// TwinCAT 3 PLC project ExternControl
// ProgramVersion: 3.1.4026.26
// libraries:
//   Tc2_Standard, * (Beckhoff Automation GmbH)
//   Tc2_System, * (Beckhoff Automation GmbH)
//   Tc2_Utilities, * (Beckhoff Automation GmbH)
// project tree:
//   APPLICATION/DISPENSER/types/ ST_DISPENSER_AXIS_PARAMETER.TcDUT, ST_DISPENSER_JOB_PARAMETER.TcDUT, ST_DISPENSER_PARAMETER.TcDUT, ST_DISPENSER_VALVES.TcDUT
//   APPLICATION/ GVL_APPLICATION.TcGVL
//   APPLICATION/JOB_CONTROL/ fb_JobBase.TcPOU, fb_JobCtrl.TcPOU
//   APPLICATION/JOB_CONTROL/types/ E_JOB_CTRL.TcDUT, E_JOB_STATE.TcDUT, E_M_FUNC.TcDUT, E_R_PARAMETER.TcDUT, E_JOB_CHECK.TcDUT, ST_AXIS_GROUP_INFO.TcDUT, ST_JOB_CTRL.TcDUT, ST_JOB_PARAMETER.TcDUT, ST_JOB_STATE.TcDUT, ST_PROG_PARAMETER.TcDUT, ST_R_ProgParameter.TcDUT, ST_TUPEL_XYZ.TcDUT
//   / GlobalTextList.TcGTLO, MAIN.TcPOU, PlcTask.TcTTO (not stored), Visualization Manager.TcVMO (not stored)
//   MAPPING/ MAPPING_out.TcPOU, MAPPING_in.TcPOU
//   MAPPING/types/ U_AXIS_CTRL.TcDUT (not stored), U_AXIS_GEAR_IN.TcDUT (not stored), U_AXIS_HOMING.TcDUT, U_AXIS_INFO.TcDUT, U_AXIS_MOTION_OPTIONS.TcDUT (not stored), U_AXIS_MOVE_DATA.TcDUT, U_AXIS_NC_PARAMETER_RD.TcDUT (not stored), U_AXIS_NC_PARAMETER_WRT.TcDUT (not stored), U_AXIS_STATE.TcDUT, U_CAM_CTRL.TcDUT, U_CAM_DATA.TcDUT, U_CAM_INFO.TcDUT (not stored), U_CAM_STATE.TcDUT, U_NCI_AXIS_ID_GROUP.TcDUT, U_NCI_CTRL.TcDUT, U_NCI_INDEX_GROUP.TcDUT (not stored), U_NCI_R_PARAMETER_I.TcDUT, U_NCI_R_PARAMETER_Q.TcDUT, U_NCI_STATE.TcDUT (not stored), U_TOUCH_PROBE_CTRL.TcDUT (not stored), U_TOUCH_PROBE_STATE.TcDUT, U_TRIGGER_CTRL.TcDUT (not stored), U_TRIGGER_STATE.TcDUT
//   PLC_MOTION/CAM/ GVL_CAM.TcGVL
//   PLC_MOTION/CAM/types/ ST_CAM_CTRL.TcDUT (not stored), ST_CAM_DATA.TcDUT, ST_CAM_INFO.TcDUT, ST_CAM_OPTIONS.TcDUT, ST_CAM_READ_VALUES_PARAMETER.TcDUT (not stored), ST_CAM_SCALING_DATA.TcDUT (not stored), ST_CAM_STATE.TcDUT, ST_MOTION_FUNCTION.TcDUT (not stored), ST_MOTION_FUNCTION_POINT.TcDUT
//   PLC_MOTION/FUNCTIONS/ GVL_FUNCTIONS.TcGVL
//   PLC_MOTION/FUNCTIONS/TOUCH_PROBE/types/ ST_2BIT.TcDUT, ST_CTRL_TOUCH_PROBE.TcDUT (not stored), ST_DC_Input.TcDUT (not stored), ST_MTI_INPUT.TcDUT (not stored), ST_MTI_STATUS.TcDUT (not stored), ST_STATE_TOUCH_PROBE.TcDUT (not stored)
//   PLC_MOTION/FUNCTIONS/TRIGGER_BOX/types/ ST_CTRL_TRIGGER.TcDUT (not stored), ST_DC_Output.TcDUT, ST_DC_State.TcDUT, ST_STATE_TRIGGER.TcDUT, T_TriggerControlBits.TcDUT
//   PLC_MOTION/NCI/ GVL_NCI.TcGVL
//   PLC_MOTION/NCI/types/ E_NCI_CHANNEL_ERROR.TcDUT, E_NCI_CTRL.TcDUT, E_NCI_INTERPRETER_STATE.TcDUT (not stored), E_NCI_STATE.TcDUT, ST_3D_Group.TcDUT (not stored), ST_Index_Group.TcDUT, ST_Interface_Group.TcDUT, ST_NciChannel_Ref.TcDUT (not stored), ST_NCI_CTRL.TcDUT (not stored), ST_NCI_M_FUNC.TcDUT (not stored), ST_NCI_STATE.TcDUT, ST_R_Parameter.TcDUT (not stored)
//   PLC_MOTION/NC_PTP/ GVL_AXIS.TcGVL (not stored)
//   PLC_MOTION/NC_PTP/types/axis/ E_AxisEncoderType.TcDUT (not stored), ST_HomeParams.TcDUT (not stored), ST_HomingOptionsExt.TcDUT (not stored)
//   PLC_MOTION/NC_PTP/types/control/ E_AXIS_CTRL.TcDUT, E_AXIS_STATE.TcDUT, ST_AXIS_CTRL.TcDUT (not stored), ST_AXIS_INFO.TcDUT (not stored), ST_AXIS_STATE.TcDUT, ST_GEAR_IN.TcDUT (not stored), ST_HOMING.TcDUT, ST_MOTION_OPTIONS.TcDUT, ST_MOVE_DATA.TcDUT (not stored), ST_NC_PARAMETER.TcDUT
//   PLC_MOTION/_GVL/ PLC_CONSTANT.TcGVL (not stored)
//   XTS_TRANSPORT/ GVL_XTS_CONSTANTS.TcGVL
//   _DUT/ f_GetProgress.TcPOU (not stored), f_GetState.TcPOU (not stored), E_CHECK_STATE.TcDUT (not stored), E_PROGRESS.TcDUT (not stored)
//   _MSG/class/ fb_LocalTime.TcPOU, fb_MessageData.TcPOU, fb_MessageDataCtrl.TcPOU
//   _MSG/ f_MessageSet.TcPOU, GVL_MSG_AXIS.TcGVL, GVL_MSG_XTS.TcGVL, I_MessageData.TcIO
//   _MSG/types/ e_Device.TcDUT, E_MessageType.TcDUT, E_MESSAGE_BATCH.TcDUT (not stored), E_MESSAGE_CHECK.TcDUT, E_MESSAGE_CTRL.TcDUT (not stored), E_MESSAGE_FLOW.TcDUT, E_MESSAGE_STATE.TcDUT (not stored), e_Subdevice.TcDUT, ST_Message.TcDUT (not stored), ST_MESSAGE_CTRL.TcDUT (not stored), ST_MESSAGE_STATE.TcDUT (not stored), TL_E_MESSAGETYPE.TcTLO
//   _XML/Configuration/ fb_Configuration.TcPOU
//   _XML/Configuration/types/ ST_Configuration.TcDUT, ST_CONFIG_DISPENSER.TcDUT, ST_CONFIG_JOBS.TcDUT, ST_CONFIG_PORTAL.TcDUT
//   _XML/ fb_XmlBase.TcPOU
//   _XML/types/ E_DATA_CHECK.TcDUT (not stored), E_DATA_CTRL.TcDUT (not stored), E_DATA_STATE.TcDUT (not stored), fb_XmlRead.TcPOU (not stored), fb_XmlWrite.TcPOU (not stored), ST_DATA_CTRL.TcDUT (not stored), ST_DATA_STATE.TcDUT (not stored)
// real-time tasks:
//   TASK PlcTask: cycle T#1ms, priority 20, ADS port 350
// motion (NC):
//   TASK NC-Task 1 SAF: cycle T#2ms, priority 4, ADS port 501
//   TASK NC-Task 1 SVB: cycle T#10ms, priority 8, ADS port 511
//   AXIS AxisX (id 1)
//     OtherSettings: AllowMotionCmdToSlave=true
//     encoder EncType=1
//     drive DrvType=5
//       Analog: TorqueSetpointScale=10, ScaleFactorActTorque=0.1
//       TimeComp: TaskDelayCycles=1
//     controller CtrType=1
//       CtrPara: PriorControlFactor=1
//         Observer: BandWidth=20
//   AXIS AxisY (id 2)
//     OtherSettings: AllowMotionCmdToSlave=true
//     encoder EncType=1
//     drive DrvType=5
//       Analog: TorqueSetpointScale=10, ScaleFactorActTorque=0.1
//       TimeComp: TaskDelayCycles=1
//     controller CtrType=1
//       CtrPara: PriorControlFactor=1
//         Observer: BandWidth=20
//   AXIS AxisZ (id 3)
//     OtherSettings: AllowMotionCmdToSlave=true
//     encoder EncType=1
//     drive DrvType=5
//       Analog: TorqueSetpointScale=10, ScaleFactorActTorque=0.1
//       TimeComp: TaskDelayCycles=1
//     controller CtrType=1
//       CtrPara: PriorControlFactor=1
//         Observer: BandWidth=20
//   AXIS Dos_A1 (id 4)
//     OtherSettings: AllowMotionCmdToSlave=true
//     encoder EncType=1
//     drive DrvType=5
//       Analog: TorqueSetpointScale=10, ScaleFactorActTorque=0.1
//       TimeComp: TaskDelayCycles=1
//     controller CtrType=1
//       CtrPara: PriorControlFactor=1
//         Observer: BandWidth=20
//   AXIS Dos_A2 (id 5)
//     OtherSettings: AllowMotionCmdToSlave=true
//     encoder EncType=1
//     drive DrvType=5
//       Analog: TorqueSetpointScale=10, ScaleFactorActTorque=0.1
//       TimeComp: TaskDelayCycles=1
//     controller CtrType=1
//       CtrPara: PriorControlFactor=1
//         Observer: BandWidth=20
//   AXIS Axis 6 (id 6)
//     OtherSettings: AllowMotionCmdToSlave=true
//     encoder EncType=1
//     drive DrvType=5
//       Analog: TorqueSetpointScale=10, ScaleFactorActTorque=0.1
//       TimeComp: TaskDelayCycles=1
//     controller CtrType=1
//       CtrPara: PriorControlFactor=1
//         Observer: BandWidth=20
// variable links:
//   ExternControl/ExternControl Instance <-> PLC_MOTION/PLC_MOTION Instance
//     PlcTask Inputs/MAIN.eInitPlcMotion <-> PlcTask Outputs/MAIN_AXIS.eInit
//     PlcTask Inputs/MAPPING_in.AxisInfo.byState <-> PlcTask Outputs/MAPPING_AXIS_out.AxisInfo.byState
//     PlcTask Inputs/MAPPING_in.AxisParameterRd.byState <-> PlcTask Outputs/MAPPING_AXIS_out.AxisParameterOut.byState
//     PlcTask Inputs/MAPPING_in.AxisState.byState <-> PlcTask Outputs/MAPPING_AXIS_out.AxisState.byState
//     PlcTask Inputs/MAPPING_in.CamInfo.byState <-> PlcTask Outputs/MAPPING_AXIS_out.CamInfo.byState
//     PlcTask Inputs/MAPPING_in.CamState.byState <-> PlcTask Outputs/MAPPING_AXIS_out.CamState.byState
//     PlcTask Inputs/MAPPING_in.NciRparameters.byState <-> PlcTask Outputs/MAPPING_AXIS_out.NciRparameters.byCtrl
//     PlcTask Inputs/MAPPING_in.NciState.byState <-> PlcTask Outputs/MAPPING_AXIS_out.NciState.byState
//     PlcTask Inputs/MAPPING_in.TouchState.byState <-> PlcTask Outputs/MAPPING_AXIS_out.TouchProbeState.byState
//     PlcTask Inputs/MAPPING_in.TriggerState.byState <-> PlcTask Outputs/MAPPING_AXIS_out.TriggerState.byState
//     PlcTask Outputs/MAPPING_out.AxisCtrl.byCtrl <-> PlcTask Inputs/MAPPING_AXIS_in.AxisCtrl.byCtrl
//     PlcTask Outputs/MAPPING_out.AxisGearInData.byCtrl <-> PlcTask Inputs/MAPPING_AXIS_in.AxisGearInData.byCtrl
//     PlcTask Outputs/MAPPING_out.AxisHoming.byCtrl <-> PlcTask Inputs/MAPPING_AXIS_in.AxisHoming.byCtrl
//     PlcTask Outputs/MAPPING_out.AxisMotionOptions.byCtrl <-> PlcTask Inputs/MAPPING_AXIS_in.AxisMotionOptions.byCtrl
//     PlcTask Outputs/MAPPING_out.AxisMoveData.byCtrl <-> PlcTask Inputs/MAPPING_AXIS_in.AxisMoveData.byCtrl
//     PlcTask Outputs/MAPPING_out.AxisParameterWrt.byCtrl <-> PlcTask Inputs/MAPPING_AXIS_in.AxisParameterIn.byCtrl
//     PlcTask Outputs/MAPPING_out.CamCtrl.byCtrl <-> PlcTask Inputs/MAPPING_AXIS_in.CamControl.byCtrl
//     PlcTask Outputs/MAPPING_out.CamData.byCtrl <-> PlcTask Inputs/MAPPING_AXIS_in.CamData.byCtrl
//     PlcTask Outputs/MAPPING_out.NciAxisGroup.byCtrl <-> PlcTask Inputs/MAPPING_AXIS_in.NciAxisGroup.byCtrl
//     PlcTask Outputs/MAPPING_out.NciControl.byCtrl <-> PlcTask Inputs/MAPPING_AXIS_in.NciControl.byCtrl[1]
//     PlcTask Outputs/MAPPING_out.NciRparameters.byCtrl <-> PlcTask Inputs/MAPPING_AXIS_in.NciRparameters.byCtrl
//     PlcTask Outputs/MAPPING_out.TouchCtrl.byCtrl <-> PlcTask Inputs/MAPPING_AXIS_in.TouchProbeControl.byCtrl
//     PlcTask Outputs/MAPPING_out.TriggerCtrl.byCtrl <-> PlcTask Inputs/MAPPING_AXIS_in.TriggerControl.byCtrl
//   PLC_MOTION/PLC_MOTION Instance <-> NC-Task 1 SAF/Axes/Axis 6
//     PlcTask Inputs/GVL_AXIS.AxisRef[6].NcToPlc <-> Outputs/ToPlc
//     PlcTask Outputs/GVL_AXIS.AxisRef[6].PlcToNc <-> Inputs/FromPlc
//   PLC_MOTION/PLC_MOTION Instance <-> NC-Task 1 SAF/Axes/AxisX
//     PlcTask Inputs/GVL_AXIS.AxisRef[1].NcToPlc <-> Outputs/ToPlc
//     PlcTask Outputs/GVL_AXIS.AxisRef[1].PlcToNc <-> Inputs/FromPlc
//   PLC_MOTION/PLC_MOTION Instance <-> NC-Task 1 SAF/Axes/AxisY
//     PlcTask Inputs/GVL_AXIS.AxisRef[2].NcToPlc <-> Outputs/ToPlc
//     PlcTask Outputs/GVL_AXIS.AxisRef[2].PlcToNc <-> Inputs/FromPlc
//   PLC_MOTION/PLC_MOTION Instance <-> NC-Task 1 SAF/Axes/AxisZ
//     PlcTask Inputs/GVL_AXIS.AxisRef[3].NcToPlc <-> Outputs/ToPlc
//     PlcTask Outputs/GVL_AXIS.AxisRef[3].PlcToNc <-> Inputs/FromPlc
//   PLC_MOTION/PLC_MOTION Instance <-> NC-Task 1 SAF/Axes/Dos_A1
//     PlcTask Inputs/GVL_AXIS.AxisRef[4].NcToPlc <-> Outputs/ToPlc
//     PlcTask Outputs/GVL_AXIS.AxisRef[4].PlcToNc <-> Inputs/FromPlc
//   PLC_MOTION/PLC_MOTION Instance <-> NC-Task 1 SAF/Axes/Dos_A2
//     PlcTask Inputs/GVL_AXIS.AxisRef[5].NcToPlc <-> Outputs/ToPlc
//     PlcTask Outputs/GVL_AXIS.AxisRef[5].PlcToNc <-> Inputs/FromPlc
//   PLC_MOTION/PLC_MOTION Instance <-> NC-Task 1 SAF/Channel XYZ
//     PlcTask Inputs/GVL_NCI.NciCtrl[1]._stChannelRef.NcToPlc <-> Outputs/ToPlc
//     PlcTask Outputs/GVL_NCI.NciCtrl[1]._stChannelRef.PlcToNc <-> Inputs/FromPlc

// ---- APPLICATION/DISPENSER/types/ST_DISPENSER_AXIS_PARAMETER.TcDUT
TYPE ST_DISPENSER_AXIS_PARAMETER :
STRUCT
  // configuration data for dispenser axis
  AxisIndex       : UINT;   // gfbAxisController[] index for PLC MOTION LAYER
  PistonDiameter  : LREAL :=   2.0;   // diameter for volume calc
  PistonArea      : LREAL :=  PI;     // (PistonDiameter/2)² * PI
  LimitUpper      : LREAL :=  10.0;   // upper limit of axis
  LimitLower      : LREAL :=   0.0;   // lower limit of axis
  LimitVelo       : LREAL :=  50.0;   // max dispensing velocity --> material constant
  LimitAccDec     : LREAL := 500.0;   // max dynamic --> material constant
END_STRUCT
END_TYPE

// ---- APPLICATION/DISPENSER/types/ST_DISPENSER_JOB_PARAMETER.TcDUT
TYPE ST_DISPENSER_JOB_PARAMETER :
STRUCT
  Volume    : LREAL := 10.0;      // [mm³]
  Velocity  : LREAL := 10.0;      // [mm³/s]
  AccDec    : LREAL := 100.0;     // [mm³/s²]
  tDelay    : TIME  := T#10MS;    // [ms]
END_STRUCT
END_TYPE

// ---- APPLICATION/DISPENSER/types/ST_DISPENSER_PARAMETER.TcDUT
TYPE ST_DISPENSER_PARAMETER :
STRUCT
  Component           : UINT  := 1;       // 1 or 2 component dispenser
  ValveInDelay        : TIME  := T#10MS;  // switch time for infeed valves  [ms]
  ValveOutDelay       : TIME  := T#10MS;  // switch time for outfeed valves [ms]

  AxisParameter       : ARRAY[1..GVL_APPLICATION.MAX_DISPENSER_COMPONENT] OF ST_DISPENSER_AXIS_PARAMETER;
END_STRUCT
END_TYPE

// ---- APPLICATION/DISPENSER/types/ST_DISPENSER_VALVES.TcDUT
TYPE ST_DISPENSER_VALVES :
STRUCT
  PistonCheck   AT %I*    : ARRAY[1..MAX_DISPENSER_COMPONENT] OF BOOL; // Piston contact with axis
  Infeed        AT %Q*    : ARRAY[1..MAX_DISPENSER_COMPONENT] OF BOOL; // infeed  valve control
  Outfeed       AT %Q*    : ARRAY[1..MAX_DISPENSER_COMPONENT] OF BOOL; // outfeed valve control
END_STRUCT
END_TYPE

// ---- APPLICATION/JOB_CONTROL/types/E_JOB_CTRL.TcDUT
{attribute 'qualified_only'}
{attribute 'strict'}
{attribute 'to_string'}
TYPE E_JOB_CTRL :
(
	JOB_NULL,
  JOB_INIT    := 10,
  JOB_IDLE,
  JOB_RESET,
  JOB_HOME,
  JOB_RINSE,
  JOB_AUTO    := 20
)UINT;
END_TYPE

// ---- APPLICATION/JOB_CONTROL/types/E_JOB_STATE.TcDUT
{attribute 'qualified_only'}
//{attribute 'strict'}
{attribute 'to_string'}
TYPE E_JOB_STATE :
(
	JOB_NULL,
  JOB_INIT    := 10,
  JOB_IDLE,
  JOB_RESET,
  JOB_HOME,
  JOB_RINSE,
  JOB_AUTO    := 20
)UINT;
END_TYPE

// ---- APPLICATION/JOB_CONTROL/types/E_M_FUNC.TcDUT
{attribute 'qualified_only'}
TYPE E_M_FUNC :
(
  //---------------------------------------------------------------------------
  // NCI --> PLC
  // m-functions
  // enumeration for NCI M functions with project specific meaning
  //---------------------------------------------------------------------------
  // reserved M functions for NCI 2, 17, 30
	E_NO_FUNC,
  E_PROG_END          :=  2,
  E_PROG_SUB_END      := 17,
  E_PROG_ALL_END      := 30,

  // used in project, defined in MOTION NC-Task ChannelXYZ.Interpreter.M-Functions
  E_AXIS_STARTUP_POSITION     := 101, // NCI has moved  to startup position (AM/AM)
  E_AXIS_WAIT_START           := 102, // NCI is waiting at startup position (BM/BM)
  E_AXIS_WAIT_END             := 103, // NCI is waiting after last G code expression (AM/AM)
  E_PROG_WAIT_END             := 104, // nc file is done
  //---------------------------------------------------------------------------

  //---------------------------------------------------------------------------
  // m-function handshakes by using m-function pairs
  //---------------------------------------------------------------------------
  E_PROG_DISP_FILL            := 150, // NCI-->PLC, fill dispenser with volume R_PROG_DISPENSER_FILL
  E_PROG_DISP_FILL_DONE       := 151, // PLC-->NCI, handshake from PLC, dispenser is filled

  E_PROG_DISP_OUT_START       := 152, // NCI-->PLC, start dispenser axis
  E_PROG_DISP_OUT_WORKING     := 153, // PLC-->NCI, dispenser axis were started --> now move on
  E_PROG_DISP_OUT_DONE        := 154  // PLC-->NCI, dispenser axis is at low position 
)UINT;
END_TYPE

// ---- APPLICATION/JOB_CONTROL/types/E_R_PARAMETER.TcDUT
{attribute 'qualified_only'}
{attribute 'strict'}
TYPE E_R_PARAMETER :
(
	R_START_POS_X         := 900,
  R_START_POS_Y,
  R_START_POS_Z,
  R_PROG_SAFE_Z         := 905,

  R_PROG_DISPENSER_WORKING_DELAY := 907,  // time dispenser delays feedback on start of dispensing axis
  R_PROG_DISPENSER_FILL := 908,  // intake volume for dispenser, corresponding M func --> E_PROG_DISP_FILL (start fill) --> E_PROG_DISP_FILL_DONE (handshake for fill done, now axis may move on)
  R_PROG_DISPENSER_VELO := 909   // requested dispensing velocity by GST-Code !rSet(909, <value>)


);
END_TYPE

// ---- APPLICATION/JOB_CONTROL/types/E_JOB_CHECK.TcDUT
{attribute 'qualified_only'}
{attribute 'strict'}
{attribute 'to_string'}
TYPE E_JOB_CHECK :
(
  CHECK_NULL,

  POINTER_NULL                        :=  9000,
  POINTER_NULL_UNIT_CTRL,
  POINTER_NULL_UNIT_STATE,

  POINTER_NULL_AXIS_CTRL              :=  9010,
  POINTER_NULL_AXIS_STATE,
  POINTER_NULL_AXIS_INFO,
  POINTER_NULL_AXIS_MOVE_DATA,
  POINTER_NULL_AXIS_INDEX,
  POINTER_NULL_AXIS_IDENTITY,

  POINTER_NULL_NCI_CHN_CTRL           :=  9020,
  POINTER_NULL_NCI_CHN_STATE,

  POINTER_NULL_JOB_PARAMETER          :=  9030,

  POINTER_NULL_SCALE_COM_CONTROL      :=  9040,
  POINTER_NULL_SCALE_COM_STATE,
  POINTER_NULL_SCALE_CONFIG,

  AXIS_RANGE_START_INVALID            :=  9100,
  AXIS_RANGE_END_INVALID,
  AXIS_DISPENSER_COMPONENTS_INVALID,

  NCI_CONFIGURATION_INVALID           :=  9200,
  CHANNEL_INDEX_INVALID,
  NCI_R_PARAMETER_INVALID,
  NCI_FILE_CTRL_INVALID,
  NCI_FILE_STATE_INVALID,

  POINTER_NULL_HOME_PARAMETER         :=  9300,
  POINTER_NULL_RINSE_PARAMETER,
  POINTER_NULL_WEIGH_PARAMETER,
  POINTER_NULL_MEAS_PARAMETER,
  POINTER_NULL_AUTO_PARAMETER,
  POINTER_NULL_STRIP_PARAMETER,

  POINTER_NULL_DISPENSER_PARAMETER    :=  9310,

  INTERFACE_NULL                      :=  9900,
  INTERFACE_NULL_UNIT_CTRL,
  INTERFACE_NULL_DISPENSER,

  CHECK_DONE                          := 10000

)UINT;
END_TYPE

// ---- APPLICATION/JOB_CONTROL/types/ST_AXIS_GROUP_INFO.TcDUT
TYPE ST_AXIS_GROUP_INFO :
STRUCT
  // result structure for searching NC Axis ID in global array of axis
  nAxisId         : UDINT;  // TwinCAT NC AxisId
  nAxisIndex      : UDINT;  // index in global axis array

  bHasValue       : BIT;    // plausibility check for nAxisId > 0
  bValid          : BIT;    // ID search did lead to an index (input ID == 0 --> not bValid)
  bMainAxis       : BIT;    // main axis (X,Y,Z)
END_STRUCT
END_TYPE

// ---- APPLICATION/JOB_CONTROL/types/ST_JOB_CTRL.TcDUT
TYPE ST_JOB_CTRL :
STRUCT
  Cmd         : E_JOB_CTRL;
END_STRUCT
END_TYPE

// ---- APPLICATION/JOB_CONTROL/types/ST_JOB_PARAMETER.TcDUT
TYPE ST_JOB_PARAMETER :
STRUCT
  Position        : ST_TUPEL_XYZ;
  // z-axis value for collision free movement of X,Y; used prior to movement of X,Y
  CollisionZ      : LREAL;               

  // dynamic parameters for movement of axis; 1 = X, 2 = Y, 3 = Z
  DynConstraint   : ARRAY[1..3] OF ST_MOVE_DATA;

  // how much, how fast shall be dispensed
  Dispenser       : ST_DISPENSER_JOB_PARAMETER; 
END_STRUCT
END_TYPE

// ---- APPLICATION/JOB_CONTROL/types/ST_JOB_STATE.TcDUT
TYPE ST_JOB_STATE :
STRUCT
  State         : E_JOB_STATE;
END_STRUCT
END_TYPE

// ---- APPLICATION/JOB_CONTROL/types/ST_PROG_PARAMETER.TcDUT
{attribute 'pack_mode' := '2'}
TYPE ST_PROG_PARAMETER :
STRUCT
  sFilename                   : STRING(255) := 'Test_GST.nc';

  stRParameter                : ST_R_ProgParameter;

END_STRUCT
END_TYPE

// ---- APPLICATION/JOB_CONTROL/types/ST_R_ProgParameter.TcDUT
{attribute 'pack_mode' := '2'}
TYPE ST_R_ProgParameter :
STRUCT
  _nStart               : DINT := 900;
  _nCount               : DINT := 10;
  _rRParamsWrite        : ARRAY[0..MAX_R_PARA] OF LREAL;
  _rRParamsRead         : ARRAY[0..MAX_R_PARA] OF LREAL;
END_STRUCT
END_TYPE

// ---- APPLICATION/JOB_CONTROL/types/ST_TUPEL_XYZ.TcDUT
TYPE ST_TUPEL_XYZ :
STRUCT
  x : LREAL;
  y : LREAL;
  z : LREAL;
END_STRUCT
END_TYPE

// ---- MAPPING/types/U_AXIS_HOMING.TcDUT
TYPE U_AXIS_HOMING :
UNION

  stCtrl              : ARRAY[1..MAX_AXIS] OF ST_HOMING;

  byCtrl    AT %Q*    : ARRAY[1..MAX_AXIS] OF
                        ARRAY[1..SIZEOF(ST_HOMING)] OF BYTE;
END_UNION
END_TYPE

// ---- MAPPING/types/U_AXIS_INFO.TcDUT
TYPE U_AXIS_INFO :
UNION

  stState             : ARRAY[1..MAX_AXIS] OF ST_AXIS_INFO;

  byState  AT %I*     : ARRAY[1..MAX_AXIS] OF
                        ARRAY[1..SIZEOF(ST_AXIS_INFO)] OF BYTE;
END_UNION
END_TYPE

// ---- MAPPING/types/U_AXIS_MOVE_DATA.TcDUT
TYPE U_AXIS_MOVE_DATA :
UNION

  stCtrl              : ARRAY[1..MAX_AXIS] OF ST_MOVE_DATA;

  byCtrl    AT %Q*    : ARRAY[1..MAX_AXIS] OF
                        ARRAY[1..SIZEOF(ST_MOVE_DATA)] OF BYTE;
END_UNION
END_TYPE

// ---- MAPPING/types/U_AXIS_STATE.TcDUT
TYPE U_AXIS_STATE :
UNION

  stState             : ARRAY[1..MAX_AXIS] OF ST_AXIS_STATE;

  byState   AT %I*    : ARRAY[1..MAX_AXIS] OF
                        ARRAY[1..SIZEOF(ST_AXIS_STATE)] OF BYTE;
END_UNION
END_TYPE

// ---- MAPPING/types/U_CAM_CTRL.TcDUT
TYPE U_CAM_CTRL :
UNION
  stCtrl              : ARRAY[1..MAX_AXIS] OF ST_CAM_CTRL;

  byCtrl    AT %q*    : ARRAY[1..MAX_AXIS] OF
                        ARRAY[1..SIZEOF(ST_CAM_CTRL)] OF BYTE;
END_UNION
END_TYPE

// ---- MAPPING/types/U_CAM_DATA.TcDUT
TYPE U_CAM_DATA :
UNION
  stCtrl              : ARRAY[1..MAX_AXIS] OF ST_CAM_DATA;

  byCtrl    AT %q*    : ARRAY[1..MAX_AXIS] OF
                        ARRAY[1..SIZEOF(ST_CAM_DATA)] OF BYTE;
END_UNION
END_TYPE

// ---- MAPPING/types/U_CAM_STATE.TcDUT
TYPE U_CAM_STATE :
UNION
  stState             : ARRAY[1..MAX_AXIS] OF ST_CAM_STATE;

  byState   AT %i*    : ARRAY[1..MAX_AXIS] OF
                        ARRAY[1..SIZEOF(ST_CAM_STATE)] OF BYTE;
END_UNION
END_TYPE

// ---- MAPPING/types/U_NCI_AXIS_ID_GROUP.TcDUT
TYPE U_NCI_AXIS_ID_GROUP :
UNION

  stCtrl              : ARRAY[1..MAX_NCI_CH] OF ST_3D_Group;

  byCtrl    AT %q*    : ARRAY[1..MAX_NCI_CH] OF
                        ARRAY[1..SIZEOF(ST_3D_Group)] OF BYTE;
END_UNION
END_TYPE

// ---- MAPPING/types/U_NCI_CTRL.TcDUT
TYPE U_NCI_CTRL :
UNION

  stCtrl              : ARRAY[1..MAX_NCI_CH] OF ST_NCI_CTRL;

  byCtrl    AT %q*    : ARRAY[1..MAX_NCI_CH] OF
                        ARRAY[1..SIZEOF(ST_NCI_CTRL)] OF BYTE;
END_UNION
END_TYPE

// ---- MAPPING/types/U_NCI_R_PARAMETER_I.TcDUT
TYPE U_NCI_R_PARAMETER_I :
UNION

  stState             : ARRAY[1..MAX_NCI_CH] OF ST_R_Parameter;

  byState   AT %I*    : ARRAY[1..MAX_NCI_CH] OF
                        ARRAY[1..SIZEOF(ST_R_Parameter)] OF BYTE;
END_UNION
END_TYPE

// ---- MAPPING/types/U_NCI_R_PARAMETER_Q.TcDUT
TYPE U_NCI_R_PARAMETER_Q :
UNION

  stCtrl              : ARRAY[1..MAX_NCI_CH] OF ST_R_Parameter;

  byCtrl    AT %Q*    : ARRAY[1..MAX_NCI_CH] OF
                        ARRAY[1..SIZEOF(ST_R_Parameter)] OF BYTE;
END_UNION
END_TYPE

// ---- MAPPING/types/U_TOUCH_PROBE_STATE.TcDUT
TYPE U_TOUCH_PROBE_STATE :
UNION
  stState              : ARRAY[1..MAX_TOUCH_PROBE] OF ST_STATE_TOUCH_PROBE;

  byState    AT %i*   : ARRAY[1..MAX_TOUCH_PROBE] OF
                        ARRAY[1..SIZEOF(ST_STATE_TOUCH_PROBE)] OF BYTE;
END_UNION
END_TYPE

// ---- MAPPING/types/U_TRIGGER_STATE.TcDUT
TYPE U_TRIGGER_STATE :
UNION
  stState              : ARRAY[1..MAX_TRIGGER_BOX] OF ST_STATE_TRIGGER;

  byState    AT %i*   : ARRAY[1..MAX_TRIGGER_BOX] OF
                        ARRAY[1..SIZEOF(ST_STATE_TRIGGER)] OF BYTE;
END_UNION
END_TYPE

// ---- PLC_MOTION/CAM/types/ST_CAM_DATA.TcDUT
{attribute 'pack_mode' := '2'}
TYPE ST_CAM_DATA :
STRUCT
  // MC_CamInfo_V2 parameters
  bAtMasterPosition       : BIT;    // If AtMasterPosition is TRUE, the data related to the specified MasterPosition is determined. Otherwise the data refers to the current master position.
  nMasterIndex            : UINT;   // Index in GVL_AXIS.AxisRef[nMasterIndex]

  rMasterPosition         : LREAL;  // Master position to which the data that is determined refers. This input parameter is not necessary if AtMasterPosition is FALSE.
  rActivationPosition     : LREAL;
  nActivationMode         : UINT;

  nCamTableId             : UDINT;  // For multi-cam plate coupling, the CamTableId also has to be transferred explicitly. If a single cam plate is involved in the coupling, the CamTableId can be set to 0.
  nPointId                : UDINT;
  nPointIndex             : UDINT;  // index of MotionFunction array
  nNumPoints              : UDINT;  // 0 = full motion function size

  stReadValuesParameter   : ST_CAM_READ_VALUES_PARAMETER;

  stCamScalingData        : ST_CAM_SCALING_DATA;
  stOptions               : ST_CAM_OPTIONS;
END_STRUCT
END_TYPE

// ---- PLC_MOTION/CAM/types/ST_CAM_INFO.TcDUT
{attribute 'pack_mode' := '2'}
TYPE ST_CAM_INFO :
STRUCT
  bPeriodic                     : BIT;
  bMasterAbsolute               : BIT;
  bSlaveAbsolute                : BIT;
  bScalingPending               : BIT;
  bCamDataQueued                : BIT;
  bCamTableQueued               : BIT;

  nTableType                    : INT;
  nInterpolationType            : UINT;
  nNumberOfRows                 : UINT;
  nNumberOfColumns              : UINT;
  nMasterAxisId                 : UINT;
  nSlaveAxisId                  : UINT;

  rMasterCamStartPos            : LREAL; (* Master pos. of the first cam table point (raw, unscaled cam table pos.) *)
  rSlaveCamStartPos             : LREAL; (* Slave pos. of the first cam table point (raw, unscaled cam table pos.) *)
  rRawMasterPeriod              : LREAL; (* raw, unscaled difference between last and first cam point *)
  rRawSlaveStroke               : LREAL; (* raw, unscaled difference between last and first cam point *)
  rMasterAxisCouplingPos        : LREAL; (* Master axis position when slave has been coupled *)
  rSlaveAxisCouplingPos         : LREAL; (* Slave axis position when slave has been coupled *)

  rMasterOffset                 : LREAL; (* total master offset *)
  rSlaveOffset                  : LREAL; (* total slave offset *)
  rMasterScaling                : LREAL; (* total master scaling factor *)
  rSlaveScaling                 : LREAL; (* total slave scaling factor *)
  rSumOfSlaveStrokes            : LREAL; (* sum of the slave strokes up to ActualMasterAxisPos *)
  rSumOfSuperpositionDistance   : LREAL; (* sum of additional moves through MC_MoveSuperimposed *)
  rActualMasterAxisPos          : LREAL; (* absolute set position of the master axis *)
  rActualSlaveAxisPos           : LREAL; (* absolute set position of the slave axis *)
  rActualMasterCamPos           : LREAL; (* raw, unscaled cam table position of the master *)
  rActualSlaveCamPos            : LREAL; (* raw, unscaled cam table position of the slave *)
  rActualPhaseShift             : LREAL;

  nScalingActivationMode        : UINT;
  rScalingActivationPos         : LREAL;
  nScalingMasterScalingMode     : UINT;
  nScalingSlaveScalingMode      : UINT;
  
  nOnlineChangeActivationMode   : UINT;
  rOnlineChangeActivationPos    : LREAL;
  nOnlineChangeMasterScalingMode: UINT;
  nOnlineChangeSlaveScalingMode : UINT;
  
  nCamExchangeCamTableID        : UDINT;
  nCamExchangeActivationMode    : UINT;
  rCamExchangeActivationPos     : LREAL;
  nCamExchangeMasterScalingMode : UINT;
  nCamExchangeSlaveScalingMode  : UINT;
END_STRUCT
END_TYPE

// ---- PLC_MOTION/CAM/types/ST_CAM_OPTIONS.TcDUT
{attribute 'pack_mode' := '2'}
TYPE ST_CAM_OPTIONS :
STRUCT
  nInterpolationType      : UINT;
  nCamOperationMode       : UINT;
  nReferenceCamTableId    : UDINT;
END_STRUCT
END_TYPE

// ---- PLC_MOTION/CAM/types/ST_CAM_STATE.TcDUT
{attribute 'pack_mode' := '2'}
TYPE ST_CAM_STATE :
STRUCT
  bError              : BIT;

  eState              : E_AXIS_STATE; // mirror the requested command + E_PROGRESS

  wCamCouplingState   : ARRAY[0..7] OF WORD;
  nCamCouplingTableId : ARRAY[0..7] OF UINT;

  nNumPointsRead      : UDINT;
END_STRUCT
END_TYPE

// ---- PLC_MOTION/CAM/types/ST_MOTION_FUNCTION_POINT.TcDUT
{attribute 'pack_mode' := '2'}
TYPE ST_MOTION_FUNCTION_POINT :
STRUCT
   nPointIndex            : UINT;
   nFunctionType          : UINT;
   wPointType             : WORD;
   nRelIndexNextPoint     : UINT;
   rMasterPos             : LREAL; (* X *)
   rSlavePos              : LREAL; (* Y *)
   rSlaveVelo             : LREAL; (* Y' *)
   rSlaveAcc              : LREAL; (* Y'' *)
   rSlaveJerk             : LREAL; (* Y''' *)
END_STRUCT
END_TYPE

// ---- PLC_MOTION/FUNCTIONS/TOUCH_PROBE/types/ST_2BIT.TcDUT
TYPE ST_2BIT :
STRUCT
  b1  : BIT;
  b2  : BIT;
END_STRUCT
END_TYPE

// ---- PLC_MOTION/FUNCTIONS/TRIGGER_BOX/types/ST_DC_Output.TcDUT
TYPE ST_DC_Output :
STRUCT
   dcStartTime      : ULINT;   (*64 bit next Action time of EL2252*)
   nActivate        : BYTE;
   Ch1_Output       : BOOL;
   Ch1_Tristate     : BOOL;
   Ch2_Output       : BOOL;
   Ch2_Tristate     : BOOL;
END_STRUCT
END_TYPE

// ---- PLC_MOTION/FUNCTIONS/TRIGGER_BOX/types/ST_DC_State.TcDUT
TYPE ST_DC_State :
STRUCT
  SysTime     : ULINT;
  {attribute 'displaymode':='binary'}
  Feedback    : USINT; // Bit 0: Output 1
                       // Bit 1: Tristate 1
                       // Bit 2: Output 2
                       // Bit 3: Tristate 2
END_STRUCT
END_TYPE

// ---- PLC_MOTION/FUNCTIONS/TRIGGER_BOX/types/ST_STATE_TRIGGER.TcDUT
TYPE ST_STATE_TRIGGER :
STRUCT
  State           : UINT; // 0 := deactivated, 100 := BUSY, 1000 := DONE, 9000 := ERROR
  Init            : UINT;
  // FlashTimestamp  : ARRAY[1..GVL_FUNCTIONS.MAX_TRIGGER_COUNT] OF ULINT; // DC timestamp
  FlashPosition   : ARRAY[1..MAX_TRIGGER_COUNT] OF LREAL; // AxisPosition for DC timestamp
END_STRUCT
END_TYPE

// ---- PLC_MOTION/FUNCTIONS/TRIGGER_BOX/types/T_TriggerControlBits.TcDUT
TYPE T_TriggerControlBits :
STRUCT
  Enable        : BIT;
  Init          : BIT;
  NoFeedback    : BIT;
{attribute 'hide'} 
  b3            : BIT;
{attribute 'hide'} 
  b4            : BIT;
{attribute 'hide'} 
  b5            : BIT;
{attribute 'hide'} 
  b6            : BIT;
{attribute 'hide'} 
  b7            : BIT;
END_STRUCT
END_TYPE

// ---- PLC_MOTION/NCI/types/E_NCI_CHANNEL_ERROR.TcDUT
{attribute 'qualified_only'}
{attribute 'strict'}
TYPE E_NCI_CHANNEL_ERROR :
(
  e_Null,
  e_InvalidReference_ChannelRef,
  e_AxisConfigurationMismatch_McAxis,
  e_AxisConfigurationMismatch_AuxAxis


);
END_TYPE

// ---- PLC_MOTION/NCI/types/E_NCI_CTRL.TcDUT
{attribute 'qualified_only'}
{attribute 'strict'}
{attribute 'to_string'}
TYPE E_NCI_CTRL :
(
  NULL,
  INIT,
  IDLE,
  RESET,
  LOAD_PROG,
  FEED_TABLE,
  BUILD_GROUP,
  CLEAR_GROUP,

  START         := 10,
  STOP,
  STO_STOP,
  RESTART_STEP_ON,

  M_FUNC_QUIT   := 20,

  READ_R_PARA   := 30,
  WRITE_R_PARA  := 40

)UINT;
END_TYPE

// ---- PLC_MOTION/NCI/types/E_NCI_STATE.TcDUT
{attribute 'qualified_only'}
//{attribute 'strict'}
{attribute 'to_string'}
TYPE E_NCI_STATE :
(
  NULL,
  INIT,
  IDLE,
  RESET,
  LOAD_PROG,
  FEED_TABLE,
  BUILD_GROUP,
  CLEAR_GROUP,

  START         := 10,
  STOP,
  STO_STOP,
  RESTART_STEP_ON,

  M_FUNC_QUIT   := 20,

  READ_R_PARA   := 30,
  WRITE_R_PARA  := 40

)UINT;
END_TYPE

// ---- PLC_MOTION/NCI/types/ST_Index_Group.TcDUT
{attribute 'pack_mode' := '2'}
TYPE ST_Index_Group :
STRUCT
  nXAxisIdx     : UDINT := 1;
  nYAxisIdx     : UDINT := 2;
  nZAxisIdx     : UDINT := 3;

  nQ1AxisIdx    : UDINT;
  nQ2AxisIdx    : UDINT;
  nQ3AxisIdx    : UDINT;
  nQ4AxisIdx    : UDINT;
  nQ5AxisIdx    : UDINT;
END_STRUCT
END_TYPE

// ---- PLC_MOTION/NCI/types/ST_Interface_Group.TcDUT
{attribute 'pack_mode' := '2'}
TYPE ST_Interface_Group :
STRUCT
  I_Idx_XAxis     : I_McAxis;
  I_Idx_YAxis     : I_McAxis;
  I_Idx_ZAxis     : I_McAxis;

  I_Idx_Q1Axis    : I_McAxis;
  I_Idx_Q2Axis    : I_McAxis;
  I_Idx_Q3Axis    : I_McAxis;
  I_Idx_Q4Axis    : I_McAxis;
  I_Idx_Q5Axis    : I_McAxis;
END_STRUCT
END_TYPE

// ---- PLC_MOTION/NCI/types/ST_NCI_STATE.TcDUT
{attribute 'pack_mode' := '2'}
TYPE ST_NCI_STATE :
STRUCT
  eState        : E_NCI_STATE; // eCmd with offsets E_PROGRESS

  bMFuncReq     : BIT;  // M function request is active from channel

  nMFunc        : WORD; // number of active M function

  nItpState     : UINT; 
                         (*  Interpreter Operation State:
                            0  = Init failed
                            1  = Idle
                            2  = Ready
                            3  = Started
                            4  = Scanning
                            5  = Running
                            6  = Stay running
                            7  = Write table
                            8  = Search line
                            9  = End
                            10 = Single Step
                            11 = Aborting
                            12 = Aborted
                            13 = Fault
                            14 = Reset
                            15 = Stop
                            16 = Wait function
                            17 = Flush buffers
                          *) 

  rAxisOverride       : LREAL; // active override in cyclic NCI interface
  sProgramNameActive  : STRING(255);
END_STRUCT
END_TYPE

// ---- PLC_MOTION/NC_PTP/types/control/E_AXIS_CTRL.TcDUT
{attribute 'qualified_only'}
{attribute 'strict'}
{attribute 'to_string'}
TYPE E_AXIS_CTRL :
(
  AXIS_NULL,   // null command
  AXIS_INIT,
  AXIS_DISABLE,
  AXIS_ENABLE,

  AXIS_IDLE     := 10, // clear axis and enable
  AXIS_HOME,
  AXIS_MOVE_POS,
  AXIS_MOVE_VELO,
  AXIS_HALT,
  AXIS_STOP,
  AXIS_SEND_TO_POS,

  AXIS_RESET              := 19,
  AXIS_STARTUP            := 20,

  AXIS_MOVE_BUFFER        := 30,
  AXIS_MOVE_BUFFER_VELO,

  AXIS_PARAMETER_READ     := 40, // command for reading and writing parameter
  AXIS_PARAMETER_WRITE,
  AXIS_PARAMETER_WRITE_PERSISTENT,


  AXIS_GEAR_IN            := 50,
  AXIS_GEAR_OUT,
  AXIS_GEAR_IN_MULTIMASTER,

  CAM_INIT                := 60,
  CAM_IN,
  CAM_OUT,
  CAM_SCALING,
  CAM_INFO,
  CAM_RD_MOTION_FUNCTION,
  CAM_RD_MOTION_FUNCTION_POINT,
  CAM_RD_MOTION_FUNCTIONS_VALUES,
  CAM_WRT_MOTION_FUNCTION,
  CAM_WRT_MOTION_FUNCTION_POINT

)UINT;
END_TYPE

// ---- PLC_MOTION/NC_PTP/types/control/E_AXIS_STATE.TcDUT
{attribute 'qualified_only'}
{attribute 'to_string'}
TYPE E_AXIS_STATE :
(
  AXIS_NULL,   // null reaction to command
  AXIS_INIT,
  AXIS_DISABLE,
  AXIS_ENABLE,

  AXIS_NO_INIT  := 9,
  
  AXIS_IDLE     := 10, // clear axis and enable
  AXIS_HOME,
  AXIS_MOVE_POS,
  AXIS_MOVE_VELO,
  AXIS_HALT,
  AXIS_STOP,
  AXIS_SEND_TO_POS,

  AXIS_RESET              := 19,
  AXIS_STARTUP            := 20,

  AXIS_MOVE_BUFFER        := 30,
  AXIS_MOVE_BUFFER_VELO,

  AXIS_PARAMETER_READ     := 40, // command for reading and writing parameter
  AXIS_PARAMETER_WRITE,
  AXIS_PARAMETER_WRITE_PERSISTENT,


  AXIS_GEAR_IN            := 50,
  AXIS_GEAR_OUT,
  AXIS_GEAR_IN_MULTIMASTER,

  CAM_INIT                := 60,
  CAM_IN,
  CAM_OUT,
  CAM_SCALING,
  CAM_INFO,
  CAM_RD_MOTION_FUNCTION,
  CAM_RD_MOTION_FUNCTION_POINT,
  CAM_RD_MOTION_FUNCTIONS_VALUES,
  CAM_WRT_MOTION_FUNCTION,
  CAM_WRT_MOTION_FUNCTION_POINT

)UINT;
END_TYPE

// ---- PLC_MOTION/NC_PTP/types/control/ST_AXIS_STATE.TcDUT
{attribute 'pack_mode' := '2'}
TYPE ST_AXIS_STATE :
STRUCT
  eState        : E_AXIS_STATE; // mirror the requested command + E_PROGRESS
  eAxisEncoder  : E_AxisEncoderType;
END_STRUCT
END_TYPE

// ---- PLC_MOTION/NC_PTP/types/control/ST_HOMING.TcDUT
{attribute 'pack_mode' := '2'}
TYPE ST_HOMING :
STRUCT
  bExecute      : BIT;

  stHomingParam : ST_HomeParams;
END_STRUCT
END_TYPE

// ---- PLC_MOTION/NC_PTP/types/control/ST_MOTION_OPTIONS.TcDUT
{attribute 'pack_mode' := '2'}
TYPE ST_MOTION_OPTIONS :
STRUCT
  // in order for extern control to be 
  // fully independent of any library types
  // struct is built with base types
  eBufferMode   : UINT; //Tc2_MC2.MC_BufferMode;  // used in FB_McAxisCtrl.MoverBufferPos, MoveBufferVelo
  rDistance     : LREAL;                  // used in FB_McAxis.SendToPos; axis has to move rDistance for method to be done
END_STRUCT
END_TYPE

// ---- PLC_MOTION/NC_PTP/types/control/ST_NC_PARAMETER.TcDUT
{attribute 'pack_mode' := '2'}
TYPE ST_NC_PARAMETER :
STRUCT
  // in order for extern control to be 
  // fully independent of any library types
  // struct is built with base types
  ParameterNumber : INT; // Tc2_MC2.MC_AxisParameter
  rValue          : LREAL; // value (Bools are cast to real)
END_STRUCT
END_TYPE

// ---- _MSG/types/e_Device.TcDUT
{attribute 'to_string'}
TYPE e_Device :
(
  // txt file logging LOG_FILE
  Device_Null,                  // NULL               - not to be used
  Device_Main,                  // MAIN(PRG)          - reserved for MAIN(PRG)
  Device_MainAxis,              // MAIN_AXIS(PRG)     - reserved for MAIN_AXIS(PRG)
  Device_Nci,                   // NCI(PRG)           - reserved for NCI(PRG)
  Device_Cam,                   // CAM(PRG            - reserved for CAM(PRG)
  Device_Functions,             // FUNCTIONS(PRG)     - reserved for FUNCTIONS(PRG)
  Device_FlyingSaw,             // FLYING_SAW(PRG)    - reserved for FLYING_SAW(PRG)
  Device_MainApplication,       // MAIN_APP(PRG)

  Device_MoverSelector,         // single mover interface for xts applications
  Device_ParameterSelector,     // fb_ParameterSelector can only exist once in a project.
  Device_Configuration,         // fb_Configuration can handle multiple files therefore only one instance is required
  Device_XmlData,               // generic XML Data (e.g. persistent data)
  Device_Utilities,             // service calls to anyone you may want to talk to, the main intent is to get XPU and TcXtsIo data to the application side


  General           :=  1000,
  CaGroup           :=  2000,
  Xpu               :=  3000,
  XpuCtrl           :=  4000,
  Mover             :=  5000,
  MoverCtrl         :=  6000,
  XtsTransportUnit  :=  7000,
  XfcTriggerBox     :=  8000,
  XfcTouchProbe     :=  9000,
  XtsStation        := 10000,

  Camming           := 11000,
  NciChannel        := 12000,
  NciChannelCtrl    := 13000,
  Axis              := 14000,
  XfcAxis           := 15000,

  // txt file logging LOG_FILE_METRICS
  MetricsXts        := 16000,   //entries from xts Metrics are written into dedicated txt file (see f_MessageSet, here's the diverter)
  MetricsAxis       := 17000,   //entries from PLC_MOTION Metrics are written into dedicated txt file

  FlyingSaw         := 18000,


  // txt file logging LOG_FILE_APP
  Process           := 20000,
  ProcessListCtrl   := 21000,
  TicketListCtrl    := 22000,

  Application       := 30000,
  UnitControl       := 31000,

  // txt file logging LOG_FILE_PRODUCT - this is for you to use
  DataProduct       := 40000
)UDINT;
END_TYPE

// ---- _MSG/types/E_MessageType.TcDUT
{attribute 'strict'}
{attribute 'to_string'}
TYPE E_MessageType :
(
  //-----------------------------------------------------
  //-----------------------------------------------------
  //  message system:
  //  - errors are always calling f_MessageSet()
  //  - errors are always entered into its list
  //
  //  - message severity is set by this enum (like everywhere else)
  //
  //  - message frequency is set by this enum
  //    - IF you get above 50 stations, 
  //      writing to the file system takes time:
  //
  //    Batch: switching on metrics (> Empty) must not add cpu load, 
  //      --> so do not clutter here
  //
  //    Info:  regular flow of information (>Error / >Warning) 
  //           must not add significant cpu load, 
  //      --> so do not clutter here
  //
  //    Verbose and above:
  //    --> for small systems (< 96 mover, < 50 stations) 
  //        you may switch it on for everybody, 
  //        files get big quickly ;-)
  //
  //    --> switch on during test phase for a handful of stations
  //
  //    --> high detail logging always and for everybody
  //    --> we need somebody who transfers data more quickly
  //      --> I can offer a .NET(C#) ADS tool which collects the list.
  //          .NET application then pushes to database
  //-----------------------------------------------------
  //-----------------------------------------------------
  eMessageEmpty,    // he who is without bounds may speak
  eMessageBatch,    // he who counts words, counts numbers (Batch started, Next in Batch, Batch done)
  eMessageError,    // mine, your(')s, anybody's, let the numbers tell you
  eMessageWarning,  // I told you so
  eMessageInfo,     // A long time ago in a galaxy far, far away...
  eMessageVerbose,  // He talks a lot, doesn't he?; Yeah! He's very knowledgeable.
  eMessageSentient  // Keep them out of bright light, Don't get them wet, do not feed them after midnight!! No matter how much they beg!!
)DINT;
END_TYPE

// ---- _MSG/types/E_MESSAGE_CHECK.TcDUT
{attribute 'qualified_only'}
{attribute 'strict'}
{attribute 'to_string'}
TYPE E_MESSAGE_CHECK :
(
  // 9000 --> here comes your error
  MSG_CHECK_INVALID_POINTER             := 9000,
  MSG_CHECK_INVALID_POINTER_TIME,
  MSG_CHECK_INVALID_POINTER_LIST,
  MSG_CHECK_INVALID_POINTER_MSG_IDX,
  MSG_CHECK_INVALID_POINTER_ERR_IDX,
  MSG_CHECK_INVALID_POINTER_ROOT_FILE,
  MSG_CHECK_INVALID_POINTER_ROOT_DIR,
  MSG_CHECK_INVALID_POINTER_CTRL,
  MSG_CHECK_INVALID_POINTER_STATE,

  // 10000 --> here comes your man
  MSG_CHECK_DONE                        := 10000
)UINT;
END_TYPE

// ---- _MSG/types/E_MESSAGE_FLOW.TcDUT
{attribute 'qualified_only'}
{attribute 'strict'}
{attribute 'to_string'}
TYPE E_MESSAGE_FLOW :
(
  MSG_FLOW_INIT,
  MSG_FLOW_ROOT                 := 10,
  MSG_FLOW_ROOT_CREATE,
  MSG_FLOW_ROOT_CREATE_BUSY,
  MSG_FLOW_FOLDER,
  MSG_FLOW_FOLDER_CREATE,
  MSG_FLOW_FOLDER_CREATE_BUSY,
  MSG_FLOW_FILE_CREATE_DONE,
  MSG_FLOW_LINE_START           := 100,
  MSG_FLOW_LINE_BUILD,
  MSG_FLOW_LINE_CHECK,
  MSG_FLOW_WRITE_FILE_BUSY      := 200,
  MSG_FLOW_WRITE_FILE_END,
  MSG_FLOW_WRITE_FILE_DONE      := 1000
)UINT;
END_TYPE

// ---- _MSG/types/e_Subdevice.TcDUT
{attribute 'strict'}
{attribute 'to_string'}
TYPE e_Subdevice :
(
  // sub device for message system
  General                 :=  0,
  MainInit,
  // Motion Control FB Instances
  fbPower,
  fbReset,
  fbResetSercos,
  fbHalt,
  fbStop,                 // 5
  fbHome,
  fbJog,
  fbMoveVelocity1,
  fbMoveVelocity2,
  fbMoveAbsolute1,        // 10
  fbMoveAbsolute2,
  fbMoveEndless,
  fbMovePtP,
  fbMoveVelo,

  // CA CollisionAvoidance FB instances
  // CA group fb instances
  fbCaGroup             := 30,
  fbMoveToPosCa,
  fbSendToAbsPosCa,
  fbSendToModuloPosCa,
  fbGearInPosCa,
  fbGroupAddAxis,
  fbGroupRemoveAxis,
  fbGroupDisable,
  fbGroupEnable,
  fbGroupErrorRead,
  fbGroupStatusRead,
  fbGroupReset,
  fbGroupStop,
  fbHaltCa,
  fbSendToPos,

  fbGearIn                := 50,
  fbGearOut,
  fbGearInMultiMaster,

  fbGearInPos,
  fbGearInVelo,


  fbCamOut                := 80,
  fbCamInV2,
  fbCamScalingV2,
  fbCamInfoV2,
  fbReadMotionFunction,
  fbReadMotionFunctionPoint,
  fbReadMotionFunctionValues,
  fbWriteMotionFunction,
  fbWriteMotionFunctionPoint,
  fbSetOnlineChangeMode,

  fbReadParameter         := 100,
  fbReadBoolParameter,
  fbWriteParameter,
  fbWriteBoolParameter,
  fbWriteParameterPersistent,

  fbBuildGroup            := 200,
  fbClearGroup,
  fbLoadProg,
  fbResetItp,
  fbStartStopItp,
  fbEStopItp,             // 205
  fbStepOnAfterEStopItp,
  fbConfirmHskItp,
  fbDelDtgItp,
  fbNciFeedTablePreparation,
  fbNciFeedTable,         // 210
  fbReadLine,
  fbItpReadRParams,
  fbItpWriteRParams,
  Get_ItpState,
  Get_Error,              // 215


  XfcPositionAtTime       := 300,
  XfcTimeOfPosition,
  XfcTimeToPosition,
  XfcTimeToModuloPosition,
  XfcRecordedPosition,
  XfcTouchProbe,          // 305
  XfcTouchProbeEL1258,
  XfcTouchProbeOptions,
  XfcTriggerRef,
  XfcTriggerRef_MT,
  XfcEl1258Interface_MT,  // 310
  XfcRecordedPosition_MT,
  XfcTriggerOut,
  XfcTriggerStart,
  XfcSwitchOn_2252,
  XfcSwitchOff_2252,      // 315
  XfcInit,
  XfcLatchPosition,
  XfcWaitForPosition,

  AxisMode              := 1000,
  AxisControl,
  AxisStartUp,
  AxisCycle,
  AxisIdle,

  NciControl            := 2000,
  NciStartUp,
  NciCycle,
  NciIdle,
  NciJob,

  FlyingSawControl      := 2100,
  FlyingSawStartUp,


  StationLinkedList     := 3000,
  StationInitList,
  StationAddHead,
  StationAddTail,
  StationGetHead,
  StationRemoveHeadValue,
  StationGearInDistanceToSync,
  StationGearInSyncStart,
  StationGearInSyncMove,
  StationGearInSyncEnd,
  StationCalcInfeedPosition,

  StationControl        := 4000,
  StationState, 

  Xpu_fbEnvironment     := 5000,
  Xpu_fbProcessingUnit,
  Xpu_fbXpuPart,
  Xpu_fbXpuTrack,
  Xpu_fbMc2CaGroup,
  Xpu_fbParameterSet,
  Xpu_fbNctController,

  Xpu_fbPartModules     := 5500,

  Xpu_fbMoverXpu        := 6000,

  Xpu_fbNctBaseUnit     := 6500,

  TransportUnit_General := 7000,
  TransportUnit_Restart := 7010,
  TransportUnit_Start,
  TransportUnit_XpuInit,
  TransportUnit_StationClearOutfeed,

  CamControl            := 8000,
  CamStartUp,
  CamCycle,

  Process_StationCollector    := 11000,
  Process_ProcessCollector    := 11100,
  Process_ProcessCollector_Init,
  Process_ProcessCollector_Cycle,
  Process_ProcessCollector_Control,

  Process_LinkedList_GetHead,
  Process_LinkedList_RemoveHead,
  Process_LinkedList_AddTail,
  Process_LinkedList_CheckData,
  Process_StationQueue_Check,

  Process_LinkedList_Com              := 11200,
  Process_LinkedList_Com_Init,
  Process_LinkedList_Com_Cmd,
  Process_LinkedList_Com_AddHead,
  Process_LinkedList_Com_AddTail,
  Process_LinkedList_Com_DelHead,
  Process_LinkedList_Com_DelTail,
  Process_LinkedList_Com_GetHead,
  Process_LinkedList_Com_GetTail,


  Instance_Command              := 12000,
  Instance_ProcessConductor,
  Instance_BufferInfeed,
  Instance_Infeed,
  Instance_BufferOutfeed,
  Instance_Outfeed,
  Instance_Sender_Buffer,

  Ticket_LinkedList_Ctrl        := 12100,
  Ticket_LinkedList_Com_Init,
  Ticket_LinkedList_Com_Cmd,
  Ticket_LinkedList_Com_AddHead,
  Ticket_LinkedList_Com_AddTail,
  Ticket_LinkedList_Com_DelHead,
  Ticket_LinkedList_Com_DelTail,
  Ticket_LinkedList_Com_GetHead,
  Ticket_LinkedList_Com_GetTail,
  

  Application                 := 13000,
  Application_Check,
  Application_Clear,
  Application_Cmd,
  Application_Disable,
  Application_Enable,
  Application_Finish,
  Application_Init,
  Application_Proceed,
  Application_Work,

  JobBase           := 14_000,
  JobBase_Job,
  JobBase_Reset,
  JobBase_StartUp,

  JobControl        := 14_100,
  JobControl_Init,
  JobControl_Idle,
  JobControl_Reset,
  JobControl_Home,
  JobControl_Rinse,
  JobControl_Auto



)DINT;
END_TYPE

// ---- _XML/Configuration/types/ST_Configuration.TcDUT
TYPE ST_Configuration :
STRUCT
  PortalConfig        : ST_CONFIG_PORTAL;
  JobConfig           : ST_CONFIG_JOBS;
END_STRUCT
END_TYPE

// ---- _XML/Configuration/types/ST_CONFIG_DISPENSER.TcDUT
TYPE ST_CONFIG_DISPENSER :
STRUCT
  // axis config for volumetric dispenser
  DispenserParameter    : ST_DISPENSER_PARAMETER;
END_STRUCT
END_TYPE

// ---- _XML/Configuration/types/ST_CONFIG_JOBS.TcDUT
TYPE ST_CONFIG_JOBS :
STRUCT
  // Job descriptions, you may write the missing ones yourself
  ParameterHome         : ST_JOB_PARAMETER;
  ParameterRinse        : ST_JOB_PARAMETER;
  ParameterAuto         : ST_JOB_PARAMETER;
  ParameterStrip        : ST_JOB_PARAMETER;
END_STRUCT
END_TYPE

// ---- _XML/Configuration/types/ST_CONFIG_PORTAL.TcDUT
TYPE ST_CONFIG_PORTAL :
STRUCT
  // NCI
  // axis NC/PtP Id
  AxisIdentity          : ST_3D_Group;
END_STRUCT
END_TYPE

// ---- APPLICATION/GVL_APPLICATION.TcGVL
{attribute 'qualified_only'}
VAR_GLOBAL CONSTANT
  MAX_DISPENSER_COMPONENT       : UINT := 2;
END_VAR
VAR_GLOBAL
  //-----------------------------------------------------------------------------------------------
  // APPLICATION territory
  //-----------------------------------------------------------------------------------------------
  //-----------------------------------------------------------------------------------------------
  // NCI portal control
  //  - handles state and initialisation of NCI portal
  //  - checks NC AxisId at startup from config (ST_3D_GROUP)
  //  - Builds 3D group from config
  //  - Executes ST_JOB_PARAMETER in axis coordinates
  //    - switch on axis in 3D group
  //    - initialize NCI via ST_NCI_CTRL/ST_NCI_STATE (init sequence in PLC_MOTION)
  //    - move main axis to Job position

  fbNciUnitControl              : ARRAY[1..PLC_CONSTANT.MAX_NCI_CH] OF fb_JobCtrl;

END_VAR

// ---- PLC_MOTION/CAM/GVL_CAM.TcGVL
{attribute 'qualified_only'}
VAR_GLOBAL
  //-----------------------------------------------------------------------------
  // command and state structure
  //  - datafields for anyone to access
  //    - ADS via symbol
  //    - cyclic mapping to any other cyclic network/runtime
  //-----------------------------------------------------------------------------
  Ctrl                        : ARRAY[1..PLC_CONSTANT.MAX_AXIS] OF ST_CAM_CTRL;      // command structure to write into
  State                       : ARRAY[1..PLC_CONSTANT.MAX_AXIS] OF ST_CAM_STATE;     // state structure to read from


  //-----------------------------------------------------------------------------
  // data and info structure
  //  - parameter data fields for
  //    - Ctrl  --> Data
  //    - State --> Info
  //-----------------------------------------------------------------------------
  Info                        : ARRAY[1..PLC_CONSTANT.MAX_AXIS] OF ST_CAM_INFO;
  Data                        : ARRAY[1..PLC_CONSTANT.MAX_AXIS] OF ST_CAM_DATA;


  //-----------------------------------------------------------------------------
  // R/W datafields
  // - get your data here after read
  // - put your data here before write
  //
  //    - Motion Function
  //    - Motion Function Point
  //-----------------------------------------------------------------------------
  MotionFunction              : ARRAY[1..PLC_CONSTANT.MAX_AXIS] OF ST_MOTION_FUNCTION;
  MotionFunctionPoint         : ARRAY[1..PLC_CONSTANT.MAX_AXIS] OF ST_MOTION_FUNCTION_POINT;

END_VAR

// ---- PLC_MOTION/FUNCTIONS/GVL_FUNCTIONS.TcGVL
{attribute 'qualified_only'}
VAR_GLOBAL
  //-----------------------------------------------------------------------------------------------------------
  // TriggerBox for moving axis, set output to activate camera, get input timestamp from flash controller
  //-----------------------------------------------------------------------------------------------------------
  DigitalOutPutDCState          : ARRAY[1..MAX_TRIGGER_BOX] OF ST_DC_State;

  DigitalOutputDC               : ARRAY[1..MAX_TRIGGER_BOX] OF ST_DC_Output;
  DigitalInputDC                : ARRAY[1..MAX_TRIGGER_BOX] OF ST_DC_Input; // distributed clock digital input with timestamps positive & negative

  CtrlTrigger                   : ARRAY[1..MAX_TRIGGER_BOX] OF ST_CTRL_TRIGGER;
  StateTrigger                  : ARRAY[1..MAX_TRIGGER_BOX] OF ST_STATE_TRIGGER;


  //-----------------------------------------------------------------------------------------------------------
  // Touch Probe with moving axis, get input timestamp within axis window, get prcise position using the timestamp
  //-----------------------------------------------------------------------------------------------------------
  //DigitalInputDC    AT %I*      : ARRAY[1..MAX_TOUCH_PROBE] OF ST_DC_Input; // distributed clock digital input with timestamps positive & negative
  DigitalInput                  : ARRAY[1..MAX_TOUCH_PROBE] OF ST_MTI_INPUT;    // multi time stamp, one channel
  DigitalState                  : ARRAY[1..MAX_TOUCH_PROBE] OF ST_MTI_STATUS;   // multi time stamp status from terminal

  CtrlTouchProbe                : ARRAY[1..MAX_TOUCH_PROBE] OF ST_CTRL_TOUCH_PROBE;
  StateTouchProbe               : ARRAY[1..MAX_TOUCH_PROBE] OF ST_STATE_TOUCH_PROBE;
END_VAR

// ---- PLC_MOTION/NCI/GVL_NCI.TcGVL
{attribute 'qualified_only'}
VAR_GLOBAL
  AxisConfig                  : ARRAY[1..MAX_NCI_CH] OF ST_3D_Group;     // NC Axis Id to build NCI group

  ChannelCtrl                 : ARRAY[1..MAX_NCI_CH] OF ST_NCI_CTRL;
  ChannelState                : ARRAY[1..MAX_NCI_CH] OF ST_NCI_STATE;


{IF NOT defined (BSD)}
  {info 'PLC_MOTION_LAYER: WIN'}
  ProgramName                 : ARRAY[1..MAX_NCI_CH] OF STRING(255):= ['C:\TwinCAT\Mc\Nci\Test_GST.nc'];
{ELSE}
  {info 'PLC_MOTION_LAYER: BSD'}
  ProgramName                 : ARRAY[1..MAX_NCI_CH] OF STRING(255):= ['/usr/local/etc/TwinCAT/Mc/Nci/Test_GST.nc'];
{END_IF}

  ProgramNameActive           : ARRAY[1..MAX_NCI_CH] OF STRING(255);

  R_ParameterRead             : ARRAY[1..MAX_NCI_CH] OF ST_R_Parameter;
  R_ParameterWrite            : ARRAY[1..MAX_NCI_CH] OF ST_R_Parameter;

  M_FunctionCyclic            : ARRAY[1..MAX_NCI_CH] OF ST_NCI_M_FUNC; // scope variable for M function tests
END_VAR

// ---- XTS_TRANSPORT/GVL_XTS_CONSTANTS.TcGVL
//{attribute 'qualified_only'}
VAR_GLOBAL CONSTANT
//-----------------------------------------------------------------------------------------------------------------------------------------
//-----------------------------------------------------------------------------------------------------------------------------------------
//
//  HAUD 2026.03.15
//  - parameter list deleted (never used the parameter feature anyway), 
//    back to static global constants
//
//-----------------------------------------------------------------------------------------------------------------------------------------
//-----------------------------------------------------------------------------------------------------------------------------------------
//  Connections to XTS Utility Lib data: 
//  - suits this simple approach, 
//  - leaves you options to expand, 
//  - expansion and multiplication is not implemented here on purpose, 
//  - this project is designed to get the main ideas across, 
//  - setting up a matrix for multiple fb_Xpu instances with it, 
//    --> a second step you might want to organize from here; 
//        --> I leave the details up to you
//-----------------------------------------------------------------------------------------------------------------------------------------
//-----------------------------------------------------------------------------------------------------------------------------------------
  MAX_PROCESS         : UINT    := 2;
  MAX_MOVER           : UINT    := 1;
//   MAX_MODULE          : UINT    := TO_UINT(Tc3_XTS_Utility.TcIoXtsEnvironmentParameterList.MaxModulesPerPart);
//   MAX_PART            : UINT    := TO_UINT(Tc3_XTS_Utility.TcIoXtsEnvironmentParameterList.MaxXtsPartsPerXpu);
//   MAX_TRACK           : UINT    := TO_UINT(Tc3_XTS_Utility.TcIoXtsEnvironmentParameterList.MaxXtsTracksPerXpu);
//   MAX_GROUP           : UINT    := TO_UINT(Tc3_XTS_Utility.TcIoXtsEnvironmentParameterList.MaxXtsCaGroup);
// 
//   MAX_INFO_SERVER     : UINT    := TO_UINT(Tc3_XTS_Utility.TcIoXtsEnvironmentParameterList.MaxXtsInfoServer);
//   MAX_INFO_STATION    : UINT    := TO_UINT(Tc3_XTS_Utility.TcIoXtsEnvironmentParameterList.MaxXtsInfoStation);
//   MAX_INFO_STOP_POS   : UINT    := TO_UINT(Tc3_XTS_Utility.TcIoXtsEnvironmentParameterList.MaxXtsStopPositionsPerStation);
// 
//   MAX_PARAMETER_SET   : UINT    := TO_UINT(Tc3_XTS_Utility.TcIoXtsEnvironmentParameterList.MaxXtsParameterSet);
// 
//   MAX_NCT_BASE_UNIT   : UINT    := TO_UINT(Tc3_XTS_Utility.TcIoXtsEnvironmentParameterList.MaxXtsNctBaseUnitInterfaces);
//-----------------------------------------------------------------------------------------------------------------------------------------
//-----------------------------------------------------------------------------------------------------------------------------------------
//  XTS_TRANSPORT_LAYER
//  - project constants you will have to adjust in order to build your transport logic
//-----------------------------------------------------------------------------------------------------------------------------------------
//-----------------------------------------------------------------------------------------------------------------------------------------
  MAX_STATION         : UINT    := 4;

  MAX_STATION_NEST    : UINT    := 8;
  MAX_LIST_NODES      : UINT    := MAX_MOVER;
  MAX_MASTER          : UINT    := 1;
//-----------------------------------------------------------------------------------------------------------------------------------------
//-----------------------------------------------------------------------------------------------------------------------------------------
END_VAR

// ---- _MSG/GVL_MSG_AXIS.TcGVL
{attribute 'qualified_only'}
VAR_GLOBAL CONSTANT
  //-----------------------------------------------------------------------------
  // file paths for message system
  //  - compiler define option WIN switches to Windows file paths
  //-----------------------------------------------------------------------------
{IF NOT defined (BSD)}
  {info 'PLC_MOTION_LAYER: WIN'}
  LOG_DIR               : STRING  := 'C:\TwinCAT\#MsgFiles\';
{ELSE}
  {info 'PLC_MOTION_LAYER: BSD'}
  LOG_DIR               : STRING  := '/usr/local/etc/TwinCAT/#MsgFiles/';
{END_IF}

  LOG_FILE              : STRING  := concat(TO_STRING(TwinCAT_SystemInfoVarList._AppInfo.AdsPort), '_MSG_PLC_');
  LOG_FILE_METRIC       : STRING  := concat(TO_STRING(TwinCAT_SystemInfoVarList._AppInfo.AdsPort), '_MSG_Metrics_');

  MAX_MESSAGE           : UINT    := 200; // max entry in message list
END_VAR
VAR_GLOBAL
  //-----------------------------------------------------------------------------
  // Message System
  //  - Everybody uses f_MessageSet(ST_Message)
  //    - DECISION WHICH LIST IS MADE IN f_MessageSet !!
  //    - which list to use is determined by e_Device in your message
  //
  //  - MessageData instances are self sufficient and need only 
  //    datafield assignment for correct data-flow
  //
  //
  //-----------------------------------------------------------------------------
  //-----------------------------------------------------------------------------
  //-----------------------------------------------------------------------------
  // (ST_Message.eDevice := from Device_Null to XfcAxis)
  //-----------------------------------------------------------------------------
  MotionMessageData               : fb_MessageDataCtrl;
  MotionMessageCtrl               : st_message_ctrl;
  MotionMessageState              : st_message_state;

  MotionMessages                  : ARRAY[1..MAX_MESSAGE] OF ST_Message;
  MessageMotionIndex              : UINT := 0; // message index for base layer
  MessageMotionError              : UINT := 0; // error counter for base layer
  //-----------------------------------------------------------------------------
  //-----------------------------------------------------------------------------
  // (ST_Message.eDevice := e_Device.Metrics)
  //-----------------------------------------------------------------------------
  MetricMessageData               : fb_MessageDataCtrl;
  MetricMessageCtrl               : st_message_ctrl;
  MetricMessageState              : st_message_state;

  MetricMessages                  : ARRAY[1..MAX_MESSAGE] OF ST_Message;
  MessageMetricIndex              : UINT := 0; // message index for metrics data
  MessageMetricError              : UINT := 0; // error counter for metrics data
  //-----------------------------------------------------------------------------
  //-----------------------------------------------------------------------------
  fbLocalTime                     : fb_LocalTime;
  dtLocalTime                     : DT;
  sLocalTime                      : STRING;
  //-----------------------------------------------------------------------------
  //-----------------------------------------------------------------------------
  //-----------------------------------------------------------------------------
  //-----------------------------------------------------------------------------
{IF defined (TEST)}
  {info 'TEST logging enabled'}
  MessageLevel                    : E_MessageType := eMessageverbose; // a lot of messages
{ELSE}
  MessageLevel                    : E_MessageType := eMessageEmpty; // only errors are written into list 
{END_IF}

  MessageLevelAxisPtp             : ARRAY[1..PLC_CONSTANT.MAX_AXIS]   OF E_MessageType;
  MessageLevelAxisCam             : ARRAY[1..PLC_CONSTANT.MAX_AXIS]   OF E_MessageType;
  MessageLevelAxisFly             : ARRAY[1..PLC_CONSTANT.MAX_AXIS]   OF E_MessageType;
  MessageLevelNciChn              : ARRAY[1..PLC_CONSTANT.MAX_NCI_CH] OF E_MessageType;

  MessageLevelTriggerBox          : ARRAY[1..PLC_CONSTANT.MAX_TRIGGER_BOX]  OF E_MessageType;
  MessageLevelTouchProbe          : ARRAY[1..PLC_CONSTANT.MAX_TOUCH_PROBE]  OF E_MessageType;


  // diag data
  dbg_AxisIdxGearIn               : ARRAY[1..PLC_CONSTANT.MAX_AXIS]      OF BYTE; // diag for Axis gear in
  dbg_AxisIdxGearInMultiMaster    : ARRAY[1..PLC_CONSTANT.MAX_AXIS,1..4] OF BYTE; // diag for Axis gear in multi master
  dbg_AxisIdxCamIn                : ARRAY[1..PLC_CONSTANT.MAX_AXIS]      OF BYTE; // diag for Axis cam in
END_VAR

// ---- _MSG/GVL_MSG_XTS.TcGVL
{attribute 'qualified_only'}
VAR_GLOBAL CONSTANT
  //-----------------------------------------------------------------------------
  // file paths for message system
  //  - compiler define option WIN switches to Windows file paths
  //-----------------------------------------------------------------------------
{IF NOT defined (BSD)}
  {info 'WIN folders'}
  LOG_DIR               : STRING  := 'C:\TwinCAT\#MsgFiles\';       // delimiter at the end is mandatory!!
  CON_DIR               : STRING  := 'C:\TwinCAT\#Configuration\';  // delimiter at the end is mandatory!!
{ELSE}
  {info 'BSD folders'}
  LOG_DIR               : STRING  := '/usr/local/etc/TwinCAT/#MsgFiles/';       // delimiter at the end is mandatory!!
  CON_DIR               : STRING  := '/usr/local/etc/TwinCAT/#Configuration/';  // delimiter at the end is mandatory!!
{END_IF}

  LOG_FILE              : STRING  := 'MSG_XtsTransport_';
  LOG_FILE_APP          : STRING  := 'MSG_Application_';
  LOG_FILE_METRIC       : STRING  := 'MSG_XtsTransportMetrics_';

  MAX_MESSAGE           : UINT    := 2000; // max entry in message list
END_VAR
VAR_GLOBAL
  //-----------------------------------------------------------------------------
  // Message System
  //  - Everybody uses f_MessageSet(ST_Message)
  //    - DECISION WHICH LIST IS MADE IN f_MessageSet !!
  //    - which list to use is determined by e_Device in your message
  //
  //  - MessageData instances are self sufficient and need only 
  //    datafield assignment for correct data-flow
  //
  //
  //-----------------------------------------------------------------------------
  //-----------------------------------------------------------------------------
  //-----------------------------------------------------------------------------
  // (ST_Message.eDevice := e_Device.Application)
  //----------------------------------------------------------------------------- 
  ApplicationMessageData          : fb_MessageDataCtrl;
  ApplicationMessageCtrl          : st_message_ctrl;
  ApplicationMessageState         : st_message_state;

  ApplicationMessages             : ARRAY[1..MAX_MESSAGE] OF ST_Message;
  MessageApplicationIndex         : UINT := 0; // message index for higher layers (grouping, Instances, etc.)
  MessageApplicationError         : UINT := 0; // error counter for higher learning
  //-----------------------------------------------------------------------------
  //-----------------------------------------------------------------------------
  // (ST_Message.eDevice := from Device_Null to XfcAxis)
  //-----------------------------------------------------------------------------
  TransportMessageData            : fb_MessageDataCtrl;
  TransportMessageCtrl            : st_message_ctrl;
  TransportMessageState           : st_message_state;

  TransportMessages               : ARRAY[1..MAX_MESSAGE] OF ST_Message;
  MessageTransportIndex           : UINT := 0; // message index for base layer
  MessageTransportError           : UINT := 0; // error counter for base layer
  //-----------------------------------------------------------------------------
  //-----------------------------------------------------------------------------
  // (ST_Message.eDevice := e_Device.Metrics)
  //-----------------------------------------------------------------------------
  MetricsMessageData              : fb_MessageDataCtrl;
  MetricsMessageCtrl              : st_message_ctrl;
  MetricsMessageState             : st_message_state;

  MetricsMessages                 : ARRAY[1..MAX_MESSAGE] OF ST_Message;
  MessageMetricsIndex             : UINT := 0; // message index for metrics data
  MessageMetricsError             : UINT := 0; // error counter for metrics data
  //-----------------------------------------------------------------------------
  //-----------------------------------------------------------------------------
  // (ST_Message.eDevice := e_Device.ProductData)
  //-----------------------------------------------------------------------------
  ProductMessageData              : fb_MessageDataCtrl;   // This is for you
  ProductMessageCtrl              : st_message_ctrl;
  ProductMessageState             : st_message_state;

  ProductMessages                 : ARRAY[1..MAX_MESSAGE] OF ST_Message;
  MessageProductIndex             : UINT := 0; // message index for your product data
  MessageProductError             : UINT := 0; // error counter for your product data
  //-----------------------------------------------------------------------------
  //-----------------------------------------------------------------------------
  fbLocalTime                     : fb_LocalTime;
  dtLocalTime                     : DT;
  sLocalTime                      : STRING;
  //-----------------------------------------------------------------------------
  //-----------------------------------------------------------------------------
  //-----------------------------------------------------------------------------
  //-----------------------------------------------------------------------------
  MessageLevelXpu                 : E_MessageType;
  MessageLevelStations            : ARRAY[1..MAX_STATION] OF E_MessageType;
  MessageLevelMovers              : ARRAY[1..MAX_MOVER]   OF E_MessageType;

  MessageLevelProcess             : ARRAY[1..MAX_PROCESS] OF E_MessageType;

{IF defined (TEST)}
  {info 'TEST logging enabled'}
  MessageLevel                    : E_MessageType := eMessageinfo; // a lot of messages
{ELSE}
  MessageLevel                    : E_MessageType := eMessageEmpty; // only errors are written into list 
{END_IF}

END_VAR

// ---- _MSG/I_MessageData.TcIO
INTERFACE I_MessageData

PROPERTY DirRoot : POINTER to string(255)
SET
END_SET
END_PROPERTY

PROPERTY ErrorIndex : reference to uint
SET
END_SET
END_PROPERTY

PROPERTY FileRoot : pointer to string(255)
SET
END_SET
END_PROPERTY

PROPERTY LocalTime : pointer to DT
SET
END_SET
END_PROPERTY

PROPERTY MessageIndex : reference to uint
SET
END_SET
END_PROPERTY

PROPERTY MsgList : pointer to ARRAY[1..GVL_MSG_AXIS.MAX_MESSAGE] OF st_message
SET
END_SET
END_PROPERTY

END_INTERFACE

// ---- MAIN.TcPOU
//-----------------------------------------------------------------------------------------------------------------
// ExternControl: EXT_MOTION_CONTROL
//
// NCI EXAMPLE for controlling PLC_MOTION_LAYER
//-----------------------------------------------------------------------------------------------------------------
PROGRAM MAIN
VAR
  //---------------------------------------------------------------------------------------------------------------
  eInitPlcMotion  AT %I*  : E_PROGRESS;   // startup indicator from PLC_MOTION plc
  //---------------------------------------------------------------------------------------------------------------
  eInit                   : E_PROGRESS;   // this plc startup
  //---------------------------------------------------------------------------------------------------------------

  eStateAxis,
  eStateCam       : E_PROGRESS;

  stMsg                   : ST_Message;
  eMsgState               : e_message_state;
  eMsgProgress            : E_PROGRESS;
  eMtrState               : e_message_state;
  eMtrProgress            : E_PROGRESS;

  tIdleWriteMotion        : TIME := T#5S;
  tIdleWriteMetric        : TIME := T#5S;
  tonIdleWriteMotion      : Tc2_Standard.TON;
  tonIdleWriteMetric      : Tc2_Standard.TON;
END_VAR

//-----------------------------------------------------------------------------------------------------------------
// Local time; used for timestamps
//-----------------------------------------------------------------------------------------------------------------
GVL_MSG_AXIS.fbLocalTime();
GVL_MSG_XTS.sLocalTime                        :=
GVL_MSG_AXIS.sLocalTime                       := GVL_MSG_AXIS.fbLocalTime.LocalTimeString;
GVL_MSG_XTS.dtLocalTime                       :=
GVL_MSG_AXIS.dtLocalTime                      := GVL_MSG_AXIS.fbLocalTime.LocalTime;
//-----------------------------------------------------------------------------------------------------------------
//-----------------------------------------------------------------------------------------------------------------
// PLC_MOTION_LAYER startup check: 
//  - you may evaluate this on your own terms
//  - putting it here was convenient for me in the context of this simple example
//-----------------------------------------------------------------------------------------------------------------
//-----------------------------------------------------------------------------------------------------------------
IF NOT (eInitPlcMotion = E_PROGRESS.PROGRESS_DONE)
THEN
  RETURN;
END_IF
//-----------------------------------------------------------------------------------------------------------------
//-----------------------------------------------------------------------------------------------------------------
// NCI EXAMPLE for controlling PLC_MOTION_LAYER
//  - Init sequence for setting up / connecting the NCI
//-----------------------------------------------------------------------------------------------------------------
//-----------------------------------------------------------------------------------------------------------------
CASE eInit 
OF
  E_PROGRESS.PROGRESS_INVALID:

  E_PROGRESS.PROGRESS_INIT:


  E_PROGRESS.PROGRESS_STILL_WORKING:  // now your init is done. 
    eInit                             := E_PROGRESS.PROGRESS_DONE;
END_CASE

//-----------------------------------------------------------------------------------------------------------------
//-----------------------------------------------------------------------------------------------------------------
//-----------------------------------------------------------------------------------------------------------------
//  /logging
//    - all life is problem solving
//-----------------------------------------------------------------------------------------------------------------
GVL_MSG_AXIS.MotionMessageData.Ctrl           REF= GVL_MSG_AXIS.MotionMessageCtrl;
GVL_MSG_AXIS.MotionMessageData.State          REF= GVL_MSG_AXIS.MotionMessageState;
GVL_MSG_AXIS.MotionMessageData.MessageIndex   REF= GVL_MSG_AXIS.MessageMotionIndex;
GVL_MSG_AXIS.MotionMessageData.ErrorIndex     REF= GVL_MSG_AXIS.MessageMotionError;
GVL_MSG_AXIS.MotionMessageData.DirRoot        :=   ADR(GVL_MSG_AXIS.LOG_DIR);
GVL_MSG_AXIS.MotionMessageData.FileRoot       :=   ADR(GVL_MSG_AXIS.LOG_FILE);
GVL_MSG_AXIS.MotionMessageData.MsgList        :=   ADR(GVL_MSG_AXIS.MotionMessages);
GVL_MSG_AXIS.MotionMessageData.LocalTime      :=   ADR(GVL_MSG_AXIS.dtLocalTime);
GVL_MSG_AXIS.MotionMessageData();               

eMsgState                                     :=   f_GetState   (GVL_MSG_AXIS.MotionMessageState.State);
eMsgProgress                                  :=   f_GetProgress(GVL_MSG_AXIS.MotionMessageState.State);

CASE eMsgState
OF
  E_MESSAGE_STATE.MSG_STATE_NULL:
    CASE eMsgProgress
    OF
      E_PROGRESS.PROGRESS_INVALID,
      E_PROGRESS.PROGRESS_DONE:
        IF (GVL_MSG_AXIS.MessageMotionIndex > GVL_MSG_XTS.MAX_MESSAGE/100) OR
           (GVL_MSG_AXIS.MessageMotionError > 0)
        THEN
          GVL_MSG_AXIS.MotionMessageCtrl.Cmd  := E_MESSAGE_CTRL.MSG_CTRL_WRITE;
        ELSE
          tonIdleWriteMotion(IN := TRUE, PT:= tIdleWriteMotion);
          IF (tonIdleWriteMotion.Q)
          THEN
            GVL_MSG_AXIS.MotionMessageCtrl.Cmd:= E_MESSAGE_CTRL.MSG_CTRL_WRITE;
          END_IF
        END_IF
    END_CASE

  E_MESSAGE_STATE.MSG_STATE_WRITE:
    CASE eMsgProgress
    OF
      E_PROGRESS.PROGRESS_ERROR,
      E_PROGRESS.PROGRESS_DONE:
        tonIdleWriteMotion(IN := FALSE, PT:= tIdleWriteMotion);
        GVL_MSG_AXIS.MotionMessageCtrl.Cmd    := E_MESSAGE_CTRL.MSG_CTRL_NULL;
    END_CASE

ELSE
    CASE eMsgProgress
    OF
      E_PROGRESS.PROGRESS_DONE:
        GVL_MSG_AXIS.MotionMessageCtrl.Cmd    := E_MESSAGE_CTRL.MSG_CTRL_NULL;
    END_CASE
END_CASE
//-----------------------------------------------------------------------------------------------------------------
//  logging/
//-----------------------------------------------------------------------------------------------------------------
//-----------------------------------------------------------------------------------------------------------------
//-----------------------------------------------------------------------------------------------------------------
//  /Metrics
//-----------------------------------------------------------------------------------------------------------------
GVL_MSG_AXIS.MetricMessageData.Ctrl           REF= GVL_MSG_AXIS.MetricMessageCtrl;
GVL_MSG_AXIS.MetricMessageData.State          REF= GVL_MSG_AXIS.MetricMessageState;

GVL_MSG_AXIS.MetricMessageData.MessageIndex   REF= GVL_MSG_AXIS.MessageMetricIndex;
GVL_MSG_AXIS.MetricMessageData.ErrorIndex     REF= GVL_MSG_AXIS.MessageMetricError;

GVL_MSG_AXIS.MetricMessageData.DirRoot        :=   ADR(GVL_MSG_AXIS.LOG_DIR);
GVL_MSG_AXIS.MetricMessageData.FileRoot       :=   ADR(GVL_MSG_AXIS.LOG_FILE_METRIC);

GVL_MSG_AXIS.MetricMessageData.MsgList        :=   ADR(GVL_MSG_AXIS.MetricMessages);
GVL_MSG_AXIS.MetricMessageData.LocalTime      :=   ADR(GVL_MSG_AXIS.dtLocalTime);

GVL_MSG_AXIS.MetricMessageData();

eMtrState                                     := f_GetState   (GVL_MSG_AXIS.MetricMessageState.State);
eMtrProgress                                  := f_GetProgress(GVL_MSG_AXIS.MetricMessageState.State);

CASE eMtrState
OF
  E_MESSAGE_STATE.MSG_STATE_NULL:
    CASE eMtrProgress
    OF
      E_PROGRESS.PROGRESS_INVALID:
        IF (GVL_MSG_AXIS.MessageMetricIndex > GVL_MSG_XTS.MAX_MESSAGE/100) OR
           (GVL_MSG_AXIS.MessageMetricError > 0)
        THEN
          GVL_MSG_AXIS.MetricMessageCtrl.Cmd  := E_MESSAGE_CTRL.MSG_CTRL_WRITE;
        ELSE
          tonIdleWriteMetric(IN := TRUE, PT:= tIdleWriteMetric);
          IF (tonIdleWriteMetric.Q)
          THEN
            GVL_MSG_AXIS.MetricMessageCtrl.Cmd:= E_MESSAGE_CTRL.MSG_CTRL_WRITE;
          END_IF
        END_IF
    END_CASE

  E_MESSAGE_STATE.MSG_STATE_WRITE:
    CASE eMtrProgress
    OF
      E_PROGRESS.PROGRESS_ERROR,
      E_PROGRESS.PROGRESS_DONE:
        tonIdleWriteMetric(IN := FALSE, PT:= tIdleWriteMetric);
        GVL_MSG_AXIS.MetricMessageCtrl.Cmd    := E_MESSAGE_CTRL.MSG_CTRL_NULL;
    END_CASE
ELSE
    CASE eMtrProgress
    OF
      E_PROGRESS.PROGRESS_DONE:
        GVL_MSG_AXIS.MetricMessageCtrl.Cmd    := E_MESSAGE_CTRL.MSG_CTRL_NULL;
    END_CASE
END_CASE
//-----------------------------------------------------------------------------------------------------------------
//  Metrics/
//-----------------------------------------------------------------------------------------------------------------
//-----------------------------------------------------------------------------------------------------------------

END_PROGRAM

// ---- APPLICATION/JOB_CONTROL/fb_JobCtrl.TcPOU
//---------------------------------------------------------------------------------------------------------------
//
//  HAUD 2026.09.20
//    - PLC_MOTION_LAYER
//      - This is a Job Control instance for accessing PtP and NCI functionalities
//    - e_progress as the generic the result offset
//    - class specific check enum E_JOB_CHECK
//
//
//  fb_JobCtrl
//  - main functionblock when using XYZ-axis (PtP and NCI) with dispenser
//  - extends fb_JobBase for executing the axis movements of jobs
//  - executes PtP and NCI jobs
//  - procedure for each job: 
//    - movement and dispenser
//
//
//---------------------------------------------------------------------------------------------------------------
// This SOFTWARE is provided as an Example by THE PROVIDER "as is" and "with all faults." THE PROVIDER makes no 
// representations or warranties of any kind concerning the safety, suitability, lack of viruses, inaccuracies, 
// typographical errors, or other harmful components of this SOFTWARE. There are inherent dangers in the use of 
// any software, and you are solely responsible for determining whether this SOFTWARE is compatible with your 
// equipment and other software installed on your equipment. You are also solely responsible for the protection 
// of your equipment and backup of your data, and THE PROVIDER will not be liable for any damages you may suffer 
// in connection with using, modifying, or distributing this SOFTWARE.
//---------------------------------------------------------------------------------------------------------------
FUNCTION_BLOCK fb_JobCtrl EXTENDS fb_JobBase
VAR
  _stCtrl             : REFERENCE TO ST_JOB_CTRL;
  _stState            : REFERENCE TO ST_JOB_STATE;

  _eCmd,
  _eCmdOld            : E_JOB_CTRL;

  _eState             : E_JOB_STATE;

//  _fbGstDos           : fb_GstDos; // start of *.nc file, mFunc Handshake for dispenser start

  _stProgParameter    : ST_PROG_PARAMETER; // TODO: get data from file

  _stRParameterNCI    : REFERENCE TO ST_R_Parameter;

  _sProgCtrl,
  _sProgState         : REFERENCE TO STRING(255);

  _stConfiguration    : REFERENCE TO ST_Configuration;
END_VAR

//-----------------------------------------------------------------------------
//-----------------------------------------------------------------------------
IF NOT Check() THEN RETURN; END_IF
//-----------------------------------------------------------------------------
//-----------------------------------------------------------------------------
// get command from outside world
//-----------------------------------------------------------------------------
_eCmd                               := _stCtrl.Cmd;
//-----------------------------------------------------------------------------
//-----------------------------------------------------------------------------
//  OnChange react to command
//-----------------------------------------------------------------------------
IF (_eCmd <> _eCmdOld)
THEN
  // get busy
  _eState                           := Cmd(_eCmd); // get execution state for command

  IF (_MessageLevel > E_MessageType.eMessageInfo)
  THEN
    _stMsg.eType                    := E_MessageType.eMessageVerbose;
    _stMsg.eSubdevice               := e_Subdevice.JobControl;
    _stMsg.iErrorNumber             := _eCmdOld;
    _stMsg.sText                    := concat('_eCmdOld: ', TO_STRING(_eCmdOld));
  
    f_MessageSet(_stMsg);
  END_IF

  IF (_MessageLevel > E_MessageType.eMessageError)
  THEN
    _stMsg.eType                    := E_MessageType.eMessageInfo;
    _stMsg.eSubdevice               := e_Subdevice.JobControl;
    _stMsg.iErrorNumber             := _eState;
    _stMsg.sText                    := concat('E_JOB_CTRL. ', TO_STRING(_eCmd));
  
    f_MessageSet(_stMsg);
  END_IF

  _eCmdOld                          := _eCmd;
END_IF
//-----------------------------------------------------------------------------
//-----------------------------------------------------------------------------
//  execution result
//-----------------------------------------------------------------------------
CASE _eResult
OF
  E_PROGRESS.PROGRESS_INVALID:
    _stState.State                  := TO_UINT(E_PROGRESS.PROGRESS_ERROR);

  E_PROGRESS.PROGRESS_ERROR:
    _stState.State                  := _eState + E_PROGRESS.PROGRESS_ERROR;

  E_PROGRESS.PROGRESS_DONE:
    _stState.State                  := _eState + E_PROGRESS.PROGRESS_DONE;

ELSE
  //-----------------------------------------------------------------------------
  // execution state result to interface
  //-----------------------------------------------------------------------------
  _stState.State                    := _eState + _eResult;

  //-----------------------------------------------------------------------------
  //-----------------------------------------------------------------------------
  //  execution state for command
  //-----------------------------------------------------------------------------
  CASE _eState
  OF
    E_JOB_STATE.JOB_INIT:
      _eResult                      := Job_Init (TRUE);
    E_JOB_STATE.JOB_IDLE:
      _eResult                      := Job_Idle (TRUE);
    E_JOB_STATE.JOB_RESET:
      _eResult                      := Job_Reset(TRUE);
    E_JOB_STATE.JOB_HOME:
      _eResult                      := Job_Home (TRUE);
    E_JOB_STATE.JOB_RINSE:
      _eResult                      := Job_Rinse(TRUE);
    E_JOB_STATE.JOB_AUTO:
      _eResult                      := Job_Auto (TRUE);
  ELSE
      _eResult                      := E_PROGRESS.PROGRESS_INVALID;
  END_CASE
END_CASE

METHOD PRIVATE Check : BOOL
VAR_INST
  _eChk       : E_JOB_CHECK;
END_VAR
//---------------------------------------------------------------------------------------------------------------
//---------------------------------------------------------------------------------------------------------------
IF NOT CheckBase() THEN _eChk   := _eCheck; RETURN; END_IF
//---------------------------------------------------------------------------------------------------------------
//---------------------------------------------------------------------------------------------------------------
IF NOT __ISVALIDREF(_stCtrl)
THEN
  _eCheck                       := E_JOB_CHECK.POINTER_NULL_UNIT_CTRL;
  RETURN;
END_IF

IF NOT __ISVALIDREF(_stState)
THEN
  _eCheck                       := E_JOB_CHECK.POINTER_NULL_UNIT_STATE;
  RETURN;
END_IF

IF NOT __ISVALIDREF(_stRParameterNCI)
THEN
  _eCheck                       := E_JOB_CHECK.NCI_R_PARAMETER_INVALID;
  RETURN;
END_IF

IF NOT __ISVALIDREF(_sProgCtrl)
THEN
  _eCheck                       := E_JOB_CHECK.NCI_FILE_CTRL_INVALID;
  RETURN;
END_IF

IF NOT __ISVALIDREF(_sProgState)
THEN
  _eCheck                       := E_JOB_CHECK.NCI_FILE_STATE_INVALID;
  RETURN;
END_IF

IF NOT __ISVALIDREF(_stConfiguration)
THEN
  _eCheck                       := E_JOB_CHECK.NCI_CONFIGURATION_INVALID;
  RETURN;
END_IF

_eCheck                         := E_JOB_CHECK.CHECK_DONE;
Check                           := TRUE;
END_METHOD

METHOD PRIVATE Cmd : E_JOB_STATE
VAR_INPUT
  eCmd      : E_JOB_CTRL;
END_VAR
VAR_INST
  _est      : E_JOB_STATE;
  _ire      : E_PROGRESS;  
END_VAR

CASE eCmd
OF
  //-------------------------------------------------------------------------------------
  E_JOB_CTRL.JOB_INIT:
    _ire                          := Job_Init(FALSE);
    _est                          := E_JOB_STATE.JOB_INIT;

ELSE
  IF (_eInit <> E_PROGRESS.PROGRESS_DONE)
  THEN
    _ire                          := E_PROGRESS.PROGRESS_ERROR;
    _est                          := E_JOB_STATE.JOB_NULL;

    _stMsg.eType                  := E_MessageType.eMessageError;
    _stMsg.eDevice                := _eDeviceId;
    _stMsg.eSubdevice             := e_Subdevice.Application_Cmd;
    _stMsg.iErrorNumber           := eCmd;

    _stMsg.sText                  := 'eInit.';
    _stMsg.sText                  := concat(_stMsg.sText, TO_STRING(_eInit));
    _stMsg.sText                  := concat(_stMsg.sText, ': ');
    _stMsg.sText                  := concat(_stMsg.sText, TO_STRING(_ire));

    f_MessageSet(_stMsg);

  ELSE
    CASE eCmd
    OF
      //---------------------------------------------------------------------------------
      E_JOB_CTRL.JOB_IDLE:
        _est                      := E_JOB_STATE.JOB_IDLE;
        _ire                      := Job_Idle(FALSE);        
      //---------------------------------------------------------------------------------
      E_JOB_CTRL.JOB_RESET:
        _est                      := E_JOB_STATE.JOB_RESET;
        _ire                      := Job_Reset(FALSE);
      //---------------------------------------------------------------------------------
      E_JOB_CTRL.JOB_HOME:
        _est                      := E_JOB_STATE.JOB_HOME;
        _ire                      := Job_Home(FALSE);
      //---------------------------------------------------------------------------------
      E_JOB_CTRL.JOB_RINSE:
        _est                      := E_JOB_STATE.JOB_RINSE;
        _ire                      := Job_Rinse(FALSE);
      //---------------------------------------------------------------------------------
      E_JOB_CTRL.JOB_AUTO:
        _est                      := E_JOB_STATE.JOB_AUTO;
        _ire                      := Job_Auto(FALSE);

    //-----------------------------------------------------------------------------------
    ELSE
      _est                        := E_JOB_STATE.JOB_NULL;

      IF (eCmd = E_AXIS_CTRL.AXIS_NULL)
      THEN
        _ire                      := E_PROGRESS.PROGRESS_DONE;
      ELSE
        _ire                      := E_PROGRESS.PROGRESS_INVALID;
  
        _stMsg.eType              := E_MessageType.eMessageError;
        _stMsg.eDevice            := _eDeviceId;
        _stMsg.eSubdevice         := e_Subdevice.Application_Cmd;
        _stMsg.iErrorNumber       := eCmd;
  
        _stMsg.sText              := 'E_JOB_CTRL.';
        _stMsg.sText              := concat(_stMsg.sText, TO_STRING(eCmd));
        _stMsg.sText              := concat(_stMsg.sText, ': ');
        _stMsg.sText              := concat(_stMsg.sText, TO_STRING(_ire));

        f_MessageSet(_stMsg);
      END_IF
    END_CASE
  END_IF // _eInit
END_CASE

_eResult                          := _ire;
Cmd                               := _est;
END_METHOD

PROPERTY Configuration : reference to ST_Configuration
SET
_stConfiguration REF= Configuration;
END_SET
END_PROPERTY

PROPERTY Ctrl : reference to ST_JOB_CTRL
SET
_stCtrl REF= Ctrl;
END_SET
END_PROPERTY

METHOD Job_Auto   : E_PROGRESS
VAR_INPUT
  Execute         : BOOL;
END_VAR
VAR_INST
  _eRslt,
  _eStateError,
  _eState         : E_PROGRESS;

  _tmpFunc        : E_M_FUNC;
END_VAR
//---------------------------------------------------------------------------------------
//---------------------------------------------------------------------------------------
IF NOT Execute THEN _eState   := _eStateError     := E_PROGRESS.PROGRESS_INIT;  RETURN; END_IF
//---------------------------------------------------------------------------------------
IF NOT Check() THEN Job_Auto  := _eState          := E_PROGRESS.PROGRESS_ERROR; RETURN; END_IF
//---------------------------------------------------------------------------------------
//---------------------------------------------------------------------------------------
CASE _eState 
of
  E_PROGRESS.PROGRESS_INIT:
    IF Execute
    THEN
      _eState                 := E_PROGRESS.PROGRESS_BUSY;
      // get job data at start
      _JobData                := _stConfiguration.JobConfig.ParameterAuto;
      _eRslt                  := Unit_Job(FALSE, _JobData);   // clear method

      IF (_MessageLevel > E_MessageType.eMessageError)
      THEN
        _stMsg.eType          := E_MessageType.eMessageInfo;
        _stMsg.eSubdevice     := e_Subdevice.JobControl_Auto;
        _stMsg.iErrorNumber   := _eState;
        _stMsg.sText          := concat(': ', TO_STRING(_eState));
      
        f_MessageSet(_stMsg);
      END_IF
    END_IF
END_CASE
//---------------------------------------------------------------------------------------
//  move PtP axis
//    - X,Y,Z
//---------------------------------------------------------------------------------------
CASE _eState
OF
  E_PROGRESS.PROGRESS_BUSY:
    _eRslt                    := Unit_Job(TRUE, _JobData);
    
    IF (_eRslt = E_PROGRESS.PROGRESS_ERROR)
    THEN
      // base class did the messaging
      // exit with error
      _eStateError            := _eState;
      _eState                 := E_PROGRESS.PROGRESS_ERROR;
      _eRslt                  := Unit_Job(FALSE, _JobData);   // clear method

    ELSIF (_eRslt = E_PROGRESS.PROGRESS_DONE)
    THEN
      // move of axis to job starting positions successful
      // next states are intended for customization
      _eState                 := E_PROGRESS.PROGRESS_STARTUP;
      _eRslt                  := Unit_Job(FALSE, _JobData);   // clear method
    END_IF
END_CASE
//---------------------------------------------------------------------------------------
//---------------------------------------------------------------------------------------
CASE _eState
OF
  E_PROGRESS.PROGRESS_PREPARE:
      // simply an inexpensive placeholder to customize initialization to your needs
      _eState                 := E_PROGRESS.PROGRESS_STARTUP;
END_CASE
//---------------------------------------------------------------------------------------
//---------------------------------------------------------------------------------------
CASE _eState
OF
  E_PROGRESS.PROGRESS_STARTUP:
      // simply an inexpensive placeholder to customize initialization to your needs
      _eState                 := E_PROGRESS.PROGRESS_CHECK;
END_CASE
//---------------------------------------------------------------------------------------
//---------------------------------------------------------------------------------------
CASE _eState
OF
  E_PROGRESS.PROGRESS_CHECK:
      _eState                 := E_PROGRESS.PROGRESS_OCCUPIED;
END_CASE
//---------------------------------------------------------------------------------------
//---------------------------------------------------------------------------------------
CASE _eState
OF
  E_PROGRESS.PROGRESS_OCCUPIED:
      _eState                 := E_PROGRESS.PROGRESS_WORKING;
END_CASE
//---------------------------------------------------------------------------------------
//---------------------------------------------------------------------------------------
CASE _eState
OF
  E_PROGRESS.PROGRESS_WORKING:
    _eState                   := E_PROGRESS.PROGRESS_DONE;

    IF (_MessageLevel > E_MessageType.eMessageError)
    THEN
      _stMsg.eType            := E_MessageType.eMessageInfo;
      _stMsg.eSubdevice       := e_Subdevice.JobControl_Auto;
      _stMsg.iErrorNumber     := _eState;
      _stMsg.sText            := concat(': ', TO_STRING(_eState));
    
      f_MessageSet(_stMsg);
    END_IF
END_CASE


Job_Auto                      := _eState;
END_METHOD

METHOD Job_Home   : E_PROGRESS
VAR_INPUT
  Execute         : BOOL;
END_VAR
VAR_INST
  _eRslt,
  _eStateError,
  _eState         : E_PROGRESS;
END_VAR
//---------------------------------------------------------------------------------------
//---------------------------------------------------------------------------------------
IF NOT Execute THEN _eState   := _eStateError     := E_PROGRESS.PROGRESS_INIT;  RETURN; END_IF
//---------------------------------------------------------------------------------------
IF NOT Check() THEN Job_Home  := _eState          := E_PROGRESS.PROGRESS_ERROR; RETURN; END_IF
//---------------------------------------------------------------------------------------
//---------------------------------------------------------------------------------------
CASE _eState 
of
  E_PROGRESS.PROGRESS_INIT:
    IF Execute
    THEN
      _eState                 := E_PROGRESS.PROGRESS_BUSY;
      // get job data at start
      _JobData                := _stConfiguration.JobConfig.ParameterHome;
      _eRslt                  := Unit_Job(FALSE, _JobData);   // clear method

      IF (_MessageLevel > E_MessageType.eMessageError)
      THEN
        _stMsg.eType          := E_MessageType.eMessageInfo;
        _stMsg.eSubdevice     := e_Subdevice.JobControl_Home;
        _stMsg.iErrorNumber   := _eState;
        _stMsg.sText          := concat(': ', TO_STRING(_eState));
      
        f_MessageSet(_stMsg);
      END_IF
    END_IF
END_CASE
//---------------------------------------------------------------------------------------
//  move PtP axis
//    - X,Y,Z
//---------------------------------------------------------------------------------------
CASE _eState
OF
  E_PROGRESS.PROGRESS_BUSY:
    _eRslt                    := Unit_Job(TRUE, _JobData);
    
    IF (_eRslt = E_PROGRESS.PROGRESS_ERROR)
    THEN
      // base class did the messaging
      // exit with error
      _eStateError            := _eState;
      _eState                 := E_PROGRESS.PROGRESS_ERROR;
      _eRslt                  := Unit_Job(FALSE, _JobData);   // clear method

    ELSIF (_eRslt = E_PROGRESS.PROGRESS_DONE)
    THEN
      // move of axis to job positions successful
      // next states are intended for customization
      _eState                 := E_PROGRESS.PROGRESS_STARTUP;
      _eRslt                  := Unit_Job(FALSE, _JobData);   // clear method
    END_IF
END_CASE
//---------------------------------------------------------------------------------------
//---------------------------------------------------------------------------------------
CASE _eState
OF
  E_PROGRESS.PROGRESS_PREPARE:
      // simply an inexpensive placeholder to customize initialization to your needs
      _eState                 := E_PROGRESS.PROGRESS_STARTUP;
END_CASE
//---------------------------------------------------------------------------------------
//---------------------------------------------------------------------------------------
CASE _eState
OF
  E_PROGRESS.PROGRESS_STARTUP:
      // simply an inexpensive placeholder to customize initialization to your needs
      _eState                 := E_PROGRESS.PROGRESS_CHECK;
END_CASE
//---------------------------------------------------------------------------------------
//---------------------------------------------------------------------------------------
CASE _eState
OF
  E_PROGRESS.PROGRESS_CHECK:
      _eState                 := E_PROGRESS.PROGRESS_OCCUPIED;
END_CASE
//---------------------------------------------------------------------------------------
//---------------------------------------------------------------------------------------
CASE _eState
OF
  E_PROGRESS.PROGRESS_OCCUPIED:
      _eState                 := E_PROGRESS.PROGRESS_WORKING;
END_CASE
//---------------------------------------------------------------------------------------
//---------------------------------------------------------------------------------------
CASE _eState
OF
  E_PROGRESS.PROGRESS_WORKING:
    _eState                   := E_PROGRESS.PROGRESS_DONE;
END_CASE


Job_Home                      := _eState;
END_METHOD

METHOD Job_Idle : E_PROGRESS
VAR_INPUT
  Execute         : BOOL;
END_VAR
VAR_INST
  _eRslt,
  _eStateError,
  _eState         : E_PROGRESS;
END_VAR
//---------------------------------------------------------------------------------------
//---------------------------------------------------------------------------------------
IF NOT Execute THEN _eState   := _eStateError     := E_PROGRESS.PROGRESS_INIT;  RETURN; END_IF
//---------------------------------------------------------------------------------------
IF NOT Check() THEN Job_Idle  := _eState          := E_PROGRESS.PROGRESS_ERROR; RETURN; END_IF
//---------------------------------------------------------------------------------------
//---------------------------------------------------------------------------------------
CASE _eState 
of
  E_PROGRESS.PROGRESS_INIT:
    IF Execute
    THEN
      _eState                 := E_PROGRESS.PROGRESS_BUSY;

      IF (_MessageLevel > E_MessageType.eMessageError)
      THEN
        _stMsg.eType          := E_MessageType.eMessageInfo;
        _stMsg.eSubdevice     := e_Subdevice.JobControl_Idle;
        _stMsg.iErrorNumber   := _eState;
        _stMsg.sText          := concat(': ', TO_STRING(_eState));
      
        f_MessageSet(_stMsg);
      END_IF
    END_IF
END_CASE
//---------------------------------------------------------------------------------------
//---------------------------------------------------------------------------------------
CASE _eState
OF
  E_PROGRESS.PROGRESS_BUSY:
    _ChannelCtrl.eCmd         := E_NCI_CTRL.IDLE;
    
    IF (_ChannelState.eState = E_NCI_STATE.IDLE + E_PROGRESS.PROGRESS_ERROR)
    THEN
      // NCI channel did the messaging --> look over there or put in msg here
      // exit with error
      _eStateError            := _eState;
      _eState                 := E_PROGRESS.PROGRESS_ERROR;


    ELSIF (_ChannelState.eState = E_NCI_STATE.IDLE + E_PROGRESS.PROGRESS_DONE)
    THEN
      // idle state of NCI successful
      // next states are intended for customization
      _eState                 := E_PROGRESS.PROGRESS_STARTUP;
    END_IF
END_CASE
//---------------------------------------------------------------------------------------
//---------------------------------------------------------------------------------------
CASE _eState
OF
  E_PROGRESS.PROGRESS_PREPARE:
      // simply an inexpensive placeholder to customize initialization to your needs
      _eState                 := E_PROGRESS.PROGRESS_STARTUP;
END_CASE
//---------------------------------------------------------------------------------------
//---------------------------------------------------------------------------------------
CASE _eState
OF
  E_PROGRESS.PROGRESS_STARTUP:
      // simply an inexpensive placeholder to customize initialization to your needs
      _eState                 := E_PROGRESS.PROGRESS_CHECK;
END_CASE
//---------------------------------------------------------------------------------------
//---------------------------------------------------------------------------------------
CASE _eState
OF
  E_PROGRESS.PROGRESS_CHECK:
      _eState                 := E_PROGRESS.PROGRESS_OCCUPIED;
END_CASE
//---------------------------------------------------------------------------------------
//---------------------------------------------------------------------------------------
CASE _eState
OF
  E_PROGRESS.PROGRESS_OCCUPIED:
      _eState                 := E_PROGRESS.PROGRESS_WORKING;
END_CASE
//---------------------------------------------------------------------------------------
//---------------------------------------------------------------------------------------
CASE _eState
OF
  E_PROGRESS.PROGRESS_WORKING:
    _eState                   := E_PROGRESS.PROGRESS_DONE;

    IF (_MessageLevel > E_MessageType.eMessageError)
    THEN
      _stMsg.eType            := E_MessageType.eMessageInfo;
      _stMsg.eSubdevice       := e_Subdevice.JobControl_Idle;
      _stMsg.iErrorNumber     := _eState;
      _stMsg.sText            := concat(': ', TO_STRING(_eState));
    
      f_MessageSet(_stMsg);
    END_IF
END_CASE


Job_Idle                      := _eState;
END_METHOD

METHOD Job_Init   : E_PROGRESS
VAR_INPUT
  Execute         : BOOL;
END_VAR
VAR_INST
  _eRslt,
  _eStateError,
  _eState         : E_PROGRESS;
END_VAR
//---------------------------------------------------------------------------------------
//---------------------------------------------------------------------------------------
IF NOT Execute THEN _eState   := _eStateError     := E_PROGRESS.PROGRESS_INIT;  RETURN; END_IF
//---------------------------------------------------------------------------------------
IF NOT Check() THEN Job_Init  := _eState          := E_PROGRESS.PROGRESS_ERROR; RETURN; END_IF
//---------------------------------------------------------------------------------------
//---------------------------------------------------------------------------------------
CASE _eState 
of
  E_PROGRESS.PROGRESS_INIT:
    IF Execute
    THEN
      _eState                 := E_PROGRESS.PROGRESS_BUSY;
      _eRslt                  := Unit_StartUp(FALSE);   // clear method

      IF (_MessageLevel > E_MessageType.eMessageError)
      THEN
        _stMsg.eType          := E_MessageType.eMessageInfo;
        _stMsg.eSubdevice     := e_Subdevice.JobControl_Init;
        _stMsg.iErrorNumber   := _eState;
        _stMsg.sText          := concat(': ', TO_STRING(_eState));
      
